  MoveL (T19476) to (113.08, 116.67, 20.1) mm, rotated rx 180 ry 0 rz -180 deg; joints [1.844, 67.674, -31.296, 3.106, -36.419, -2.5]
  Call Extruder 0.32811
  MoveL (T19477) to (108.19, 107.08, 20.1) mm, rotated rx 180 ry 0 rz -180 deg; joints [1.415, 68.728, -33.274, 2.439, -35.479, -1.986]
  Call Extruder 0.03668
  MoveL (T19478) to (108.19, 105.88, 20.1) mm, rotated rx 180 ry 0 rz -180 deg; joints [1.415, 68.728, -33.274, 2.439, -35.479, -1.986]
  Call Extruder 0.02276
  MoveL (T19479) to (108.94, 105.88, 20.1) mm, rotated rx 180 ry 0 rz -180 deg; joints [1.417, 68.56, -32.958, 2.433, -35.626, -1.978]
  Set speed (150.0 mm/s)
  MoveL (T19480) to (108.6, 106.28, 20.1) mm, rotated rx 180 ry 0 rz -180 deg; joints [1.417, 68.56, -32.958, 2.433, -35.626, -1.978]
  Set speed (25.0 mm/s)
  MoveL (T19481) to (108.6, 106.28, 20.1) mm, rotated rx 180 ry 0 rz -180 deg; joints [1.846, 67.513, -30.993, 3.099, -36.56, -2.49]
  Call Extruder 0.25102
  MoveL (T19482) to (116.84, 106.28, 20.1) mm, rotated rx 180 ry 0 rz -180 deg; joints [1.846, 67.513, -30.993, 3.099, -36.56, -2.49]
  Call Extruder 0.05979
  MoveL (T19483) to (116.84, 108.25, 20.1) mm, rotated rx 180 ry 0 rz -180 deg; joints [1.848, 67.353, -30.693, 3.093, -36.7, -2.48]
  Call Extruder 0.16307
  MoveL (T19484) to (111.48, 108.25, 20.1) mm, rotated rx 180 ry 0 rz -180 deg; joints [1.848, 67.353, -30.693, 3.093, -36.7, -2.48]
  Call Extruder 0.3456
  MoveL (T19485) to (116.65, 118.34, 20.1) mm, rotated rx 180 ry 0 rz -180 deg; joints [1.848, 67.353, -30.693, 3.093, -36.7, -2.48]
  Call Extruder 0.02131
  MoveL (T19486) to (116.65, 119.04, 20.1) mm, rotated rx 180 ry 0 rz -180 deg; joints [1.418, 68.393, -32.645, 2.427, -35.772, -1.969]
  Call Extruder 0.24283
  MoveL (T19487) to (108.68, 119.04, 20.1) mm, rotated rx 180 ry 0 rz -180 deg; joints [1.418, 68.393, -32.645, 2.427, -35.772, -1.969]
  Call Extruder 0.05979
  MoveL (T19488) to (108.68, 117.08, 20.1) mm, rotated rx 180 ry 0 rz -180 deg; joints [1.418, 68.393, -32.645, 2.427, -35.772, -1.969]
  Call Extruder 0.15438
  MoveL (T19489) to (113.75, 117.08, 20.1) mm, rotated rx 180 ry 0 rz -180 deg; joints [1.42, 68.227, -32.334, 2.421, -35.918, -1.961]
  Call Extruder 0.34538
  MoveL (T19490) to (108.6, 106.98, 20.1) mm, rotated rx 180 ry 0 rz -180 deg; joints [1.42, 68.227, -32.334, 2.421, -35.918, -1.961]
  Call Extruder 0.01947
  MoveL (T19491) to (108.6, 106.34, 20.1) mm, rotated rx 180 ry 0 rz -180 deg; joints [1.42, 68.227, -32.334, 2.421, -35.918, -1.961]
  Set speed (150.0 mm/s)
  MoveL (T19492) to (108.54, 105.89, 20.1) mm, rotated rx 180 ry 0 rz -180 deg; joints [1.85, 67.194, -30.394, 3.086, -36.84, -2.471]
  Set speed (45.0 mm/s)
  Call Extruder -1.6
  MoveL (T19493) to (108.54, 105.89, 20.1) mm, rotated rx 180 ry 0 rz -180 deg; joints [1.85, 67.194, -30.394, 3.086, -36.84, -2.471]
  Set speed (120.0 mm/s)
  MoveL (T19494) to (108.54, 105.89, 20.1) mm, rotated rx 180 ry 0 rz -180 deg; joints [1.85, 67.194, -30.394, 3.086, -36.84, -2.471]
  Call Extruder -0.38
  MoveL (T19495) to (109.66, 106.33, 20.1) mm, rotated rx 180 ry 0 rz -180 deg; joints [1.852, 67.036, -30.097, 3.08, -36.979, -2.461]
  Set speed (45.0 mm/s)
  Call Extruder -0.02
  MoveL (T19496) to (109.66, 106.33, 20.1) mm, rotated rx 180 ry 0 rz -180 deg; joints [1.852, 67.036, -30.097, 3.08, -36.979, -2.461]
  Set speed (150.0 mm/s)
  MoveL (T19497) to (109.66, 106.33, 22.1) mm, rotated rx 180 ry 0 rz -180 deg; joints [1.852, 67.036, -30.097, 3.08, -36.979, -2.461]
  MoveL (T19498) to (104.34, 103.54, 22.1) mm, rotated rx 180 ry 0 rz -180 deg; joints [1.422, 68.063, -32.025, 2.415, -36.062, -1.953]
  MoveL (T19499) to (104.34, 103.54, 20.1) mm, rotated rx 180 ry 0 rz -180 deg; joints [1.422, 68.063, -32.025, 2.415, -36.062, -1.953]
  Set speed (40.0 mm/s)
  Call Extruder 2.0
  MoveL (T19500) to (104.34, 103.54, 20.1) mm, rotated rx 180 ry 0 rz -180 deg; joints [1.422, 68.063, -32.025, 2.415, -36.062, -1.953]
  Call Extruder 0.52159
  MoveL (T19501) to (121.46, 103.54, 20.1) mm, rotated rx 180 ry 0 rz -180 deg; joints [1.423, 67.899, -31.717, 2.41, -36.206, -1.945]
  Call Extruder 0.54596
  MoveL (T19502) to (121.46, 121.46, 20.1) mm, rotated rx 180 ry 0 rz -180 deg; joints [1.854, 66.879, -29.802, 3.073, -37.117, -2.451]
  Call Extruder 0.54596
  MoveL (T19503) to (103.54, 121.46, 20.1) mm, rotated rx 180 ry 0 rz -180 deg; joints [1.854, 66.879, -29.802, 3.073, -37.117, -2.451]
  Call Extruder 0.54596
  MoveL (T19504) to (103.54, 103.54, 20.1) mm, rotated rx 180 ry 0 rz -180 deg; joints [1.856, 66.722, -29.509, 3.067, -37.253, -2.442]
  Call Extruder 0.02254
  MoveL (T19505) to (104.28, 103.54, 20.1) mm, rotated rx 180 ry 0 rz -180 deg; joints [1.856, 66.722, -29.509, 3.067, -37.253, -2.442]
  Set speed (150.0 mm/s)
  MoveL (T19506) to (103.53, 103.13, 20.1) mm, rotated rx 180 ry 0 rz -180 deg; joints [1.856, 66.722, -29.509, 3.067, -37.253, -2.442]
  Set speed (40.0 mm/s)
  MoveL (T19507) to (103.53, 103.13, 20.1) mm, rotated rx 180 ry 0 rz -180 deg; joints [1.425, 67.737, -31.412, 2.404, -36.348, -1.937]
  Call Extruder 0.55858
  MoveL (T19508) to (121.87, 103.13, 20.1) mm, rotated rx 180 ry 0 rz -180 deg; joints [1.425, 67.737, -31.412, 2.404, -36.348, -1.937]
  Call Extruder 0.57077
  MoveL (T19509) to (121.87, 121.87, 20.1) mm, rotated rx 180 ry 0 rz -180 deg; joints [1.425, 67.737, -31.412, 2.404, -36.348, -1.937]
  Call Extruder 0.57077
  MoveL (T19510) to (103.13, 121.87, 20.1) mm, rotated rx 180 ry 0 rz -180 deg; joints [1.425, 67.737, -31.412, 2.404, -36.348, -1.937]
  Call Extruder 0.57077
  MoveL (T19511) to (103.13, 103.13, 20.1) mm, rotated rx 180 ry 0 rz -180 deg; joints [1.426, 67.575, -31.109, 2.399, -36.49, -1.929]
  Call Extruder 0.01036
  MoveL (T19512) to (103.47, 103.13, 20.1) mm, rotated rx 180 ry 0 rz -180 deg; joints [1.426, 67.575, -31.109, 2.399, -36.49, -1.929]
  Set speed (150.0 mm/s)
  MoveL (T19513) to (102.72, 102.81, 20.1) mm, rotated rx 180 ry 0 rz -180 deg; joints [1.827, 66.638, -29.35, 3.014, -37.326, -2.397]
  Set speed (25.0 mm/s)
  MoveL (T19514) to (102.72, 102.81, 20.1) mm, rotated rx 180 ry 0 rz -180 deg; joints [1.827, 66.638, -29.35, 3.014, -37.326, -2.397]
  Call Extruder 0.00259
  MoveL (T19515) to (102.72, 102.72, 20.1) mm, rotated rx 180 ry 0 rz -180 deg; joints [1.827, 66.638, -29.35, 3.014, -37.326, -2.397]
  Call Extruder 0.59557
  MoveL (T19516) to (122.28, 102.72, 20.1) mm, rotated rx 180 ry 0 rz -180 deg; joints [1.796, 66.558, -29.2, 2.958, -37.395, -2.351]
  Call Extruder 0.59557
  MoveL (T19517) to (122.28, 122.28, 20.1) mm, rotated rx 180 ry 0 rz -180 deg; joints [1.796, 66.558, -29.2, 2.958, -37.395, -2.351]
  Call Extruder 0.59557
  MoveL (T19518) to (102.72, 122.28, 20.1) mm, rotated rx 180 ry 0 rz -180 deg; joints [1.796, 66.558, -29.2, 2.958, -37.395, -2.351]
  Call Extruder 0.59115
  MoveL (T19519) to (102.72, 102.87, 20.1) mm, rotated rx 180 ry 0 rz -180 deg; joints [1.428, 67.414, -30.808, 2.394, -36.631, -1.921]
  Set speed (150.0 mm/s)
  MoveL (T19520) to (102.78, 102.75, 20.1) mm, rotated rx 180 ry 0 rz -180 deg; joints [1.428, 67.414, -30.808, 2.394, -36.631, -1.921]
  Set speed (45.0 mm/s)
  Call Extruder -1.6
  MoveL (T19521) to (102.78, 102.75, 20.1) mm, rotated rx 180 ry 0 rz -180 deg; joints [1.429, 67.255, -30.508, 2.388, -36.771, -1.914]
  Set speed (120.0 mm/s)
  MoveL (T19522) to (102.78, 102.75, 20.1) mm, rotated rx 180 ry 0 rz -180 deg; joints [1.429, 67.255, -30.508, 2.388, -36.771, -1.914]
  Call Extruder -0.05166
  MoveL (T19523) to (102.72, 102.72, 20.1) mm, rotated rx 180 ry 0 rz -180 deg; joints [1.429, 67.255, -30.508, 2.388, -36.771, -1.914]
  Call Extruder -0.32834
  MoveL (T19524) to (103.65, 102.72, 20.1) mm, rotated rx 180 ry 0 rz -180 deg; joints [1.765, 66.478, -29.05, 2.902, -37.464, -2.304]
  Set speed (45.0 mm/s)
  Call Extruder -0.02
  MoveL (T19525) to (103.65, 102.72, 20.1) mm, rotated rx 180 ry 0 rz -180 deg; joints [1.765, 66.478, -29.05, 2.902, -37.464, -2.304]
  Set speed (150.0 mm/s)
  MoveL (T19526) to (103.65, 102.72, 22.1) mm, rotated rx 180 ry 0 rz -180 deg; joints [1.734, 66.398, -28.9, 2.846, -37.532, -2.258]
  MoveL (T19527) to (121.34, 120.62, 22.1) mm, rotated rx 180 ry 0 rz -180 deg; joints [1.431, 67.096, -30.21, 2.383, -36.91, -1.906]
  MoveL (T19528) to (121.34, 120.62, 20.1) mm, rotated rx 180 ry 0 rz -180 deg; joints [1.431, 67.096, -30.21, 2.383, -36.91, -1.906]
  Set speed (40.0 mm/s)
  Call Extruder 2.0
  MoveL (T19529) to (121.34, 120.62, 20.1) mm, rotated rx 180 ry 0 rz -180 deg; joints [1.431, 67.096, -30.21, 2.383, -36.91, -1.906]
  Set speed (25.0 mm/s)
  MoveL (T19530) to (121.34, 120.62, 20.1) mm, rotated rx 180 ry 0 rz -180 deg; joints [1.431, 67.096, -30.21, 2.383, -36.91, -1.906]
  Call Extruder 0.02133
  MoveL (T19531) to (120.78, 121.18, 20.1) mm, rotated rx 180 ry 0 rz -180 deg; joints [1.433, 66.939, -29.915, 2.378, -37.048, -1.899]
  Call Extruder 0.01356
  MoveL (T19532) to (120.27, 121.18, 20.1) mm, rotated rx 180 ry 0 rz -180 deg; joints [1.433, 66.939, -29.915, 2.378, -37.048, -1.899]
  Call Extruder 0.03442
  MoveL (T19533) to (121.18, 120.27, 20.1) mm, rotated rx 180 ry 0 rz -180 deg; joints [1.702, 66.319, -28.752, 2.791, -37.6, -2.212]
  Call Extruder 0.01356
  MoveL (T19534) to (121.18, 119.77, 20.1) mm, rotated rx 180 ry 0 rz -180 deg; joints [1.702, 66.319, -28.752, 2.791, -37.6, -2.212]
  Call Extruder 0.0536
  MoveL (T19535) to (119.77, 121.18, 20.1) mm, rotated rx 180 ry 0 rz -180 deg; joints [1.671, 66.24, -28.604, 2.736, -37.668, -2.166]
  Call Extruder 0.01356
  MoveL (T19536) to (119.26, 121.18, 20.1) mm, rotated rx 180 ry 0 rz -180 deg; joints [1.671, 66.24, -28.604, 2.736, -37.668, -2.166]
  Call Extruder 0.07278
  MoveL (T19537) to (121.18, 119.26, 20.1) mm, rotated rx 180 ry 0 rz -180 deg; joints [1.671, 66.24, -28.604, 2.736, -37.668, -2.166]
  Call Extruder 0.01356
  MoveL (T19538) to (121.18, 118.75, 20.1) mm, rotated rx 180 ry 0 rz -180 deg; joints [1.434, 66.782, -29.62, 2.373, -37.185, -1.891]
  Call Extruder 0.09196
  MoveL (T19539) to (118.75, 121.18, 20.1) mm, rotated rx 180 ry 0 rz -180 deg; joints [1.434, 66.782, -29.62, 2.373, -37.185, -1.891]
  Call Extruder 0.01356
  MoveL (T19540) to (118.25, 121.18, 20.1) mm, rotated rx 180 ry 0 rz -180 deg; joints [1.434, 66.782, -29.62, 2.373, -37.185, -1.891]
  Call Extruder 0.11113
  MoveL (T19541) to (121.18, 118.25, 20.1) mm, rotated rx 180 ry 0 rz -180 deg; joints [1.436, 66.626, -29.328, 2.369, -37.322, -1.884]
  Call Extruder 0.01356
  MoveL (T19542) to (121.18, 117.74, 20.1) mm, rotated rx 180 ry 0 rz -180 deg; joints [1.436, 66.626, -29.328, 2.369, -37.322, -1.884]
  Call Extruder 0.13031
  MoveL (T19543) to (117.74, 121.18, 20.1) mm, rotated rx 180 ry 0 rz -180 deg; joints [1.629, 66.186, -28.502, 2.664, -37.714, -2.108]
  Call Extruder 0.01356
  MoveL (T19544) to (117.23, 121.18, 20.1) mm, rotated rx 180 ry 0 rz -180 deg; joints [1.629, 66.186, -28.502, 2.664, -37.714, -2.108]
  Call Extruder 0.14949
  MoveL (T19545) to (121.18, 117.23, 20.1) mm, rotated rx 180 ry 0 rz -180 deg; joints [1.629, 66.186, -28.502, 2.664, -37.714, -2.108]
  Call Extruder 0.01356
  MoveL (T19546) to (121.18, 116.73, 20.1) mm, rotated rx 180 ry 0 rz -180 deg; joints [1.565, 66.182, -28.494, 2.559, -37.716, -2.025]
  Call Extruder 0.16867
  MoveL (T19547) to (116.73, 121.18, 20.1) mm, rotated rx 180 ry 0 rz -180 deg; joints [1.565, 66.182, -28.494, 2.559, -37.716, -2.025]
  Call Extruder 0.01356
  MoveL (T19548) to (116.22, 121.18, 20.1) mm, rotated rx 180 ry 0 rz -180 deg; joints [1.565, 66.182, -28.494, 2.559, -37.716, -2.025]
  Call Extruder 0.03951
  MoveL (T19549) to (117.27, 120.14, 20.1) mm, rotated rx 180 ry 0 rz -180 deg; joints [1.565, 66.182, -28.494, 2.559, -37.716, -2.025]
  Call Extruder 0.0129
  MoveL (T19550) to (117.75, 120.14, 20.1) mm, rotated rx 180 ry 0 rz -180 deg; joints [1.437, 66.471, -29.037, 2.364, -37.458, -1.877]
  Call Extruder 0.0129
  MoveL (T19551) to (117.75, 119.66, 20.1) mm, rotated rx 180 ry 0 rz -180 deg; joints [1.437, 66.471, -29.037, 2.364, -37.458, -1.877]
  Call Extruder 0.13009
  MoveL (T19552) to (121.18, 116.22, 20.1) mm, rotated rx 180 ry 0 rz -180 deg; joints [1.439, 66.317, -28.748, 2.359, -37.593, -1.87]
  Call Extruder 0.01356
  MoveL (T19553) to (121.18, 115.72, 20.1) mm, rotated rx 180 ry 0 rz -180 deg; joints [1.439, 66.317, -28.748, 2.359, -37.593, -1.87]
  Call Extruder 0.13009
  MoveL (T19554) to (117.75, 119.15, 20.1) mm, rotated rx 180 ry 0 rz -180 deg; joints [1.439, 66.317, -28.748, 2.359, -37.593, -1.87]
  Call Extruder 0.01356
  MoveL (T19555) to (117.75, 118.64, 20.1) mm, rotated rx 180 ry 0 rz -180 deg; joints [1.521, 66.132, -28.4, 2.485, -37.758, -1.965]
  Call Extruder 0.13009
  MoveL (T19556) to (121.18, 115.21, 20.1) mm, rotated rx 180 ry 0 rz -180 deg; joints [1.521, 66.132, -28.4, 2.485, -37.758, -1.965]
  Call Extruder 0.01356
  MoveL (T19557) to (121.18, 114.7, 20.1) mm, rotated rx 180 ry 0 rz -180 deg; joints [1.521, 66.132, -28.4, 2.485, -37.758, -1.965]
  Call Extruder 0.13009
  MoveL (T19558) to (117.75, 118.14, 20.1) mm, rotated rx 180 ry 0 rz -180 deg; joints [1.521, 66.132, -28.4, 2.485, -37.758, -1.965]
  Call Extruder 0.00153
  MoveL (T19559) to (117.75, 118.08, 20.1) mm, rotated rx 180 ry 0 rz -180 deg; joints [1.521, 66.132, -28.4, 2.485, -37.758, -1.965]
  Call Extruder 0.00894
  MoveL (T19560) to (117.59, 117.78, 20.1) mm, rotated rx 180 ry 0 rz -180 deg; joints [1.521, 66.132, -28.4, 2.485, -37.758, -1.965]
  Call Extruder 0.13584
  MoveL (T19561) to (121.18, 114.2, 20.1) mm, rotated rx 180 ry 0 rz -180 deg; joints [1.521, 66.132, -28.4, 2.485, -37.758, -1.965]
  Call Extruder 0.01356
  MoveL (T19562) to (121.18, 113.69, 20.1) mm, rotated rx 180 ry 0 rz -180 deg; joints [1.521, 66.132, -28.4, 2.485, -37.758, -1.965]
  Call Extruder 0.14234
  MoveL (T19563) to (117.42, 117.45, 20.1) mm, rotated rx 180 ry 0 rz -180 deg; joints [1.521, 66.132, -28.4, 2.485, -37.758, -1.965]
  Call Extruder 0.01008
  MoveL (T19564) to (117.25, 117.11, 20.1) mm, rotated rx 180 ry 0 rz -180 deg; joints [1.521, 66.132, -28.4, 2.485, -37.758, -1.965]
  Call Extruder 0.14883
  MoveL (T19565) to (121.18, 113.19, 20.1) mm, rotated rx 180 ry 0 rz -180 deg; joints [1.521, 66.132, -28.4, 2.485, -37.758, -1.965]
  Call Extruder 0.01356
  MoveL (T19566) to (121.18, 112.68, 20.1) mm, rotated rx 180 ry 0 rz -180 deg; joints [1.521, 66.132, -28.4, 2.485, -37.758, -1.965]
  Call Extruder 0.15532
  MoveL (T19567) to (117.08, 116.78, 20.1) mm, rotated rx 180 ry 0 rz -180 deg; joints [1.439, 66.317, -28.748, 2.359, -37.593, -1.87]
  Call Extruder 0.01008
  MoveL (T19568) to (116.91, 116.44, 20.1) mm, rotated rx 180 ry 0 rz -180 deg; joints [1.439, 66.317, -28.748, 2.359, -37.593, -1.87]
  Call Extruder 0.16181
  MoveL (T19569) to (121.18, 112.17, 20.1) mm, rotated rx 180 ry 0 rz -180 deg; joints [1.439, 66.317, -28.748, 2.359, -37.593, -1.87]
  Call Extruder 0.01356
  MoveL (T19570) to (121.18, 111.67, 20.1) mm, rotated rx 180 ry 0 rz -180 deg; joints [1.439, 66.323, -28.759, 2.36, -37.588, -1.87]
  Call Extruder 0.1683
  MoveL (T19571) to (116.74, 116.11, 20.1) mm, rotated rx 180 ry 0 rz -180 deg; joints [1.439, 66.323, -28.759, 2.36, -37.588, -1.87]
  Call Extruder 0.01008
  MoveL (T19572) to (116.57, 115.77, 20.1) mm, rotated rx 180 ry 0 rz -180 deg; joints [1.439, 66.323, -28.759, 2.36, -37.588, -1.87]
  Call Extruder 0.1748
  MoveL (T19573) to (121.18, 111.16, 20.1) mm, rotated rx 180 ry 0 rz -180 deg; joints [1.439, 66.323, -28.759, 2.36, -37.588, -1.87]
  Call Extruder 0.01356
  MoveL (T19574) to (121.18, 110.65, 20.1) mm, rotated rx 180 ry 0 rz -180 deg; joints [1.439, 66.323, -28.759, 2.36, -37.588, -1.87]
  Call Extruder 0.18129
  MoveL (T19575) to (116.39, 115.44, 20.1) mm, rotated rx 180 ry 0 rz -180 deg; joints [1.439, 66.323, -28.759, 2.36, -37.588, -1.87]
  Call Extruder 0.01008
  MoveL (T19576) to (116.22, 115.1, 20.1) mm, rotated rx 180 ry 0 rz -180 deg; joints [1.439, 66.323, -28.759, 2.36, -37.588, -1.87]
  Call Extruder 0.18778
  MoveL (T19577) to (121.18, 110.15, 20.1) mm, rotated rx 180 ry 0 rz -180 deg; joints [1.888, 67.418, -31.218, 3.194, -36.243, -2.577]
  Call Extruder 0.01356
  MoveL (T19578) to (121.18, 109.64, 20.1) mm, rotated rx 180 ry 0 rz -180 deg; joints [1.888, 67.418, -31.218, 3.194, -36.243, -2.577]
  Call Extruder 0.19427
  MoveL (T19579) to (116.05, 114.77, 20.1) mm, rotated rx 180 ry 0 rz -180 deg; joints [1.888, 67.652, -31.254, 3.179, -36.44, -2.558]
  Call Extruder 0.01008
  MoveL (T19580) to (115.88, 114.43, 20.1) mm, rotated rx 180 ry 0 rz -180 deg; joints [1.888, 67.652, -31.254, 3.179, -36.44, -2.558]
  Call Extruder 0.20076
  MoveL (T19581) to (121.18, 109.14, 20.1) mm, rotated rx 180 ry 0 rz -180 deg; joints [1.888, 67.652, -31.254, 3.179, -36.44, -2.558]
  Call Extruder 0.01356
  MoveL (T19582) to (121.18, 108.63, 20.1) mm, rotated rx 180 ry 0 rz -180 deg; joints [1.888, 67.652, -31.254, 3.179, -36.44, -2.558]
  Call Extruder 0.20726
  MoveL (T19583) to (115.71, 114.1, 20.1) mm, rotated rx 180 ry 0 rz -180 deg; joints [1.888, 67.652, -31.254, 3.179, -36.44, -2.558]
  Call Extruder 0.01008
  MoveL (T19584) to (115.54, 113.77, 20.1) mm, rotated rx 180 ry 0 rz -180 deg; joints [1.888, 67.652, -31.254, 3.179, -36.44, -2.558]
  Call Extruder 0.21375
  MoveL (T19585) to (121.18, 108.12, 20.1) mm, rotated rx 180 ry 0 rz -180 deg; joints [1.888, 67.652, -31.254, 3.179, -36.44, -2.558]
  Call Extruder 0.01356
  MoveL (T19586) to (121.18, 107.62, 20.1) mm, rotated rx 180 ry 0 rz -180 deg; joints [1.888, 67.652, -31.254, 3.179, -36.44, -2.558]
  Call Extruder 0.22024
  MoveL (T19587) to (115.37, 113.43, 20.1) mm, rotated rx 180 ry 0 rz -180 deg; joints [1.888, 67.652, -31.254, 3.179, -36.44, -2.558]
  Call Extruder 0.01008
  MoveL (T19588) to (115.2, 113.09, 20.1) mm, rotated rx 180 ry 0 rz -180 deg; joints [1.888, 67.652, -31.254, 3.179, -36.44, -2.558]
  Call Extruder 0.22673
  MoveL (T19589) to (121.18, 107.11, 20.1) mm, rotated rx 180 ry 0 rz -180 deg; joints [1.884, 67.911, -31.74, 3.19, -36.213, -2.575]
  Call Extruder 0.01356
  MoveL (T19590) to (121.18, 106.6, 20.1) mm, rotated rx 180 ry 0 rz -180 deg; joints [1.884, 67.911, -31.74, 3.19, -36.213, -2.575]
  Call Extruder 0.23322
  MoveL (T19591) to (115.02, 112.76, 20.1) mm, rotated rx 180 ry 0 rz -180 deg; joints [1.875, 67.966, -31.843, 3.178, -36.165, -2.566]
  Call Extruder 0.01008
  MoveL (T19592) to (114.85, 112.42, 20.1) mm, rotated rx 180 ry 0 rz -180 deg; joints [1.875, 67.966, -31.843, 3.178, -36.165, -2.566]
  Call Extruder 0.23972
  MoveL (T19593) to (121.18, 106.1, 20.1) mm, rotated rx 180 ry 0 rz -180 deg; joints [1.875, 67.966, -31.843, 3.178, -36.165, -2.566]
  Call Extruder 0.01356
  MoveL (T19594) to (121.18, 105.59, 20.1) mm, rotated rx 180 ry 0 rz -180 deg; joints [1.775, 68.208, -32.297, 3.024, -35.949, -2.449]
  Call Extruder 0.12308
  MoveL (T19595) to (117.93, 108.84, 20.1) mm, rotated rx 180 ry 0 rz -180 deg; joints [1.775, 68.208, -32.297, 3.024, -35.949, -2.449]
  Call Extruder 0.01337
  MoveL (T19596) to (117.93, 109.34, 20.1) mm, rotated rx 180 ry 0 rz -180 deg; joints [2.29, 69.699, -35.098, 4.028, -34.668, -3.315]
  Call Extruder 0.01337
  MoveL (T19597) to (117.43, 109.34, 20.1) mm, rotated rx 180 ry 0 rz -180 deg; joints [2.29, 69.699, -35.098, 4.028, -34.668, -3.315]
  Call Extruder 0.10422
  MoveL (T19598) to (114.68, 112.09, 20.1) mm, rotated rx 180 ry 0 rz -180 deg; joints [2.356, 69.707, -35.112, 4.144, -34.665, -3.41]
  Call Extruder 0.01008
  MoveL (T19599) to (114.51, 111.75, 20.1) mm, rotated rx 180 ry 0 rz -180 deg; joints [2.356, 69.707, -35.112, 4.144, -34.665, -3.41]
  Call Extruder 0.09153
  MoveL (T19600) to (116.93, 109.34, 20.1) mm, rotated rx 180 ry 0 rz -180 deg; joints [2.356, 69.707, -35.112, 4.144, -34.665, -3.41]
  Call Extruder 0.01356
  MoveL (T19601) to (116.42, 109.34, 20.1) mm, rotated rx 180 ry 0 rz -180 deg; joints [3.288, 67.468, -30.908, 5.508, -36.687, -4.422]
  Call Extruder 0.07885
  MoveL (T19602) to (114.34, 111.42, 20.1) mm, rotated rx 180 ry 0 rz -180 deg; joints [3.288, 67.468, -30.908, 5.508, -36.687, -4.422]
  Call Extruder 0.01008
  MoveL (T19603) to (114.17, 111.09, 20.1) mm, rotated rx 180 ry 0 rz -180 deg; joints [3.288, 67.468, -30.908, 5.508, -36.687, -4.422]
  Call Extruder 0.06616
  MoveL (T19604) to (115.91, 109.34, 20.1) mm, rotated rx 180 ry 0 rz -180 deg; joints [3.295, 67.17, -30.349, 5.486, -36.948, -4.389]
  Call Extruder 0.01356
  MoveL (T19605) to (115.41, 109.34, 20.1) mm, rotated rx 180 ry 0 rz -180 deg; joints [3.295, 67.17, -30.349, 5.486, -36.948, -4.389]
  Call Extruder 0.05348
  MoveL (T19606) to (114, 110.75, 20.1) mm, rotated rx 180 ry 0 rz -180 deg; joints [2.938, 66.204, -28.536, 4.801, -37.766, -3.799]
  Call Extruder 0.01008
  MoveL (T19607) to (113.83, 110.42, 20.1) mm, rotated rx 180 ry 0 rz -180 deg; joints [2.938, 66.204, -28.536, 4.801, -37.766, -3.799]
  Call Extruder 0.04079
  MoveL (T19608) to (114.9, 109.34, 20.1) mm, rotated rx 180 ry 0 rz -180 deg; joints [2.938, 66.204, -28.536, 4.801, -37.766, -3.799]
  Call Extruder 0.01356
  MoveL (T19609) to (114.39, 109.34, 20.1) mm, rotated rx 180 ry 0 rz -180 deg; joints [2.938, 66.204, -28.536, 4.801, -37.766, -3.799]
  Call Extruder 0.0281
  MoveL (T19610) to (113.65, 110.08, 20.1) mm, rotated rx 180 ry 0 rz -180 deg; joints [2.818, 66.19, -28.509, 4.604, -37.771, -3.642]
  Call Extruder 0.01008
  MoveL (T19611) to (113.48, 109.75, 20.1) mm, rotated rx 180 ry 0 rz -180 deg; joints [1.815, 68.507, -32.858, 3.112, -35.689, -2.528]
  Call Extruder 0.01542
  MoveL (T19612) to (113.89, 109.34, 20.1) mm, rotated rx 180 ry 0 rz -180 deg; joints [1.815, 68.507, -32.858, 3.112, -35.689, -2.528]
  Call Extruder 0.01356
  MoveL (T19613) to (113.38, 109.34, 20.1) mm, rotated rx 180 ry 0 rz -180 deg; joints [1.866, 68.651, -33.13, 3.21, -35.564, -2.612]
  Call Extruder 0.00725
  MoveL (T19614) to (113.19, 109.53, 20.1) mm, rotated rx 180 ry 0 rz -180 deg; joints [1.866, 68.651, -33.13, 3.21, -35.564, -2.612]
  Set speed (45.0 mm/s)
  Call Extruder -1.6
  MoveL (T19615) to (113.19, 109.53, 20.1) mm, rotated rx 180 ry 0 rz -180 deg; joints [1.866, 68.651, -33.13, 3.21, -35.564, -2.612]
  Set speed (120.0 mm/s)
  MoveL (T19616) to (113.19, 109.53, 20.1) mm, rotated rx 180 ry 0 rz -180 deg; joints [1.866, 68.651, -33.13, 3.21, -35.564, -2.612]
  Call Extruder -0.09648
  MoveL (T19617) to (113.38, 109.34, 20.1) mm, rotated rx 180 ry 0 rz -180 deg; joints [1.866, 68.651, -33.13, 3.21, -35.564, -2.612]
  Call Extruder -0.18035
  MoveL (T19618) to (113.89, 109.34, 20.1) mm, rotated rx 180 ry 0 rz -180 deg; joints [1.874, 68.709, -33.238, 3.228, -35.514, -2.628]
  Call Extruder -0.10317
  MoveL (T19619) to (113.68, 109.54, 20.1) mm, rotated rx 180 ry 0 rz -180 deg; joints [1.869, 69.145, -34.057, 3.249, -35.132, -2.658]
  Set speed (45.0 mm/s)
  Call Extruder -0.02
  MoveL (T19620) to (113.68, 109.54, 20.1) mm, rotated rx 180 ry 0 rz -180 deg; joints [1.869, 69.145, -34.057, 3.249, -35.132, -2.658]
  Set speed (150.0 mm/s)
  MoveL (T19621) to (113.68, 109.54, 22.1) mm, rotated rx 180 ry 0 rz -180 deg; joints [1.869, 69.145, -34.057, 3.249, -35.132, -2.658]
  MoveL (T19622) to (117.77, 108.5, 22.1) mm, rotated rx 180 ry 0 rz -180 deg; joints [1.869, 69.145, -34.057, 3.249, -35.132, -2.658]
  MoveL (T19623) to (117.77, 108.5, 20.1) mm, rotated rx 180 ry 0 rz -180 deg; joints [1.869, 69.145, -34.057, 3.249, -35.132, -2.658]
  Set speed (40.0 mm/s)
  Call Extruder 2.0
  MoveL (T19624) to (117.77, 108.5, 20.1) mm, rotated rx 180 ry 0 rz -180 deg; joints [1.869, 69.145, -34.057, 3.249, -35.132, -2.658]
  Set speed (25.0 mm/s)
  MoveL (T19625) to (117.77, 108.5, 20.1) mm, rotated rx 180 ry 0 rz -180 deg; joints [1.869, 69.145, -34.057, 3.249, -35.132, -2.658]
  Call Extruder 0.12917
  MoveL (T19626) to (121.18, 105.08, 20.1) mm, rotated rx 180 ry 0 rz -180 deg; joints [1.869, 69.145, -34.057, 3.249, -35.132, -2.658]
  Call Extruder 0.01356
  MoveL (T19627) to (121.18, 104.58, 20.1) mm, rotated rx 180 ry 0 rz -180 deg; joints [1.869, 69.145, -34.057, 3.249, -35.132, -2.658]
  Call Extruder 0.12308
  MoveL (T19628) to (117.93, 107.83, 20.1) mm, rotated rx 180 ry 0 rz -180 deg; joints [1.873, 68.839, -33.482, 3.234, -35.4, -2.637]
  Call Extruder 0.01356
  MoveL (T19629) to (117.93, 107.32, 20.1) mm, rotated rx 180 ry 0 rz -180 deg; joints [1.873, 68.839, -33.482, 3.234, -35.4, -2.637]
  Call Extruder 0.12308
  MoveL (T19630) to (121.18, 104.07, 20.1) mm, rotated rx 180 ry 0 rz -180 deg; joints [1.873, 68.839, -33.482, 3.234, -35.4, -2.637]
  Call Extruder 0.00678
  MoveL (T19631) to (121.18, 103.82, 20.1) mm, rotated rx 180 ry 0 rz -180 deg; joints [1.873, 68.839, -33.482, 3.234, -35.4, -2.637]
  Call Extruder 0.00678
  MoveL (T19632) to (120.93, 103.82, 20.1) mm, rotated rx 180 ry 0 rz -180 deg; joints [1.873, 68.839, -33.482, 3.234, -35.4, -2.637]
  Call Extruder 0.11349
  MoveL (T19633) to (117.93, 106.81, 20.1) mm, rotated rx 180 ry 0 rz -180 deg; joints [1.873, 68.839, -33.482, 3.234, -35.4, -2.637]
  Call Extruder 0.01356
  MoveL (T19634) to (117.93, 106.31, 20.1) mm, rotated rx 180 ry 0 rz -180 deg; joints [1.873, 68.605, -33.443, 3.249, -35.206, -2.656]
  Call Extruder 0.09431
  MoveL (T19635) to (120.42, 103.82, 20.1) mm, rotated rx 180 ry 0 rz -180 deg; joints [1.652, 70.731, -37.43, 3.008, -33.337, -2.513]
  Call Extruder 0.01356
  MoveL (T19636) to (119.92, 103.82, 20.1) mm, rotated rx 180 ry 0 rz -180 deg; joints [1.652, 70.963, -37.471, 2.993, -33.527, -2.495]
  Call Extruder 0.07513
  MoveL (T19637) to (117.93, 105.8, 20.1) mm, rotated rx 180 ry 0 rz -180 deg; joints [1.652, 70.963, -37.471, 2.993, -33.527, -2.495]
  Call Extruder 0.01356
  MoveL (T19638) to (117.93, 105.3, 20.1) mm, rotated rx 180 ry 0 rz -180 deg; joints [1.652, 70.963, -37.471, 2.993, -33.527, -2.495]
  Call Extruder 0.05596
  MoveL (T19639) to (119.41, 103.82, 20.1) mm, rotated rx 180 ry 0 rz -180 deg; joints [1.652, 70.963, -37.471, 2.993, -33.527, -2.495]
  Call Extruder 0.01356
  MoveL (T19640) to (118.9, 103.82, 20.1) mm, rotated rx 180 ry 0 rz -180 deg; joints [1.652, 70.963, -37.471, 2.993, -33.527, -2.495]
  Call Extruder 0.05183
  MoveL (T19641) to (117.53, 105.19, 20.1) mm, rotated rx 180 ry 0 rz -180 deg; joints [1.652, 70.963, -37.471, 2.993, -33.527, -2.495]
  Call Extruder 0.01356
  MoveL (T19642) to (117.03, 105.19, 20.1) mm, rotated rx 180 ry 0 rz -180 deg; joints [1.652, 70.963, -37.471, 2.993, -33.527, -2.495]
  Call Extruder 0.05183
  MoveL (T19643) to (118.4, 103.82, 20.1) mm, rotated rx 180 ry 0 rz -180 deg; joints [1.652, 70.963, -37.471, 2.993, -33.527, -2.495]
  Call Extruder 0.01356
  MoveL (T19644) to (117.89, 103.82, 20.1) mm, rotated rx 180 ry 0 rz -180 deg; joints [1.652, 70.963, -37.471, 2.993, -33.527, -2.495]
  Call Extruder 0.05183
  MoveL (T19645) to (116.52, 105.19, 20.1) mm, rotated rx 180 ry 0 rz -180 deg; joints [1.652, 70.963, -37.471, 2.993, -33.527, -2.495]
  Call Extruder 0.01356
  MoveL (T19646) to (116.02, 105.19, 20.1) mm, rotated rx 180 ry 0 rz -180 deg; joints [1.396, 70.942, -37.433, 2.527, -33.535, -2.107]
  Call Extruder 0.05183
  MoveL (T19647) to (117.38, 103.82, 20.1) mm, rotated rx 180 ry 0 rz -180 deg; joints [1.396, 70.942, -37.433, 2.527, -33.535, -2.107]
  Call Extruder 0.01356
  MoveL (T19648) to (116.88, 103.82, 20.1) mm, rotated rx 180 ry 0 rz -180 deg; joints [1.467, 70.743, -37.059, 2.643, -33.712, -2.199]
  Call Extruder 0.05183
  MoveL (T19649) to (115.51, 105.19, 20.1) mm, rotated rx 180 ry 0 rz -180 deg; joints [1.467, 70.743, -37.059, 2.643, -33.712, -2.199]
  Call Extruder 0.01356
  MoveL (T19650) to (115, 105.19, 20.1) mm, rotated rx 180 ry 0 rz -180 deg; joints [1.467, 70.743, -37.059, 2.643, -33.712, -2.199]
  Call Extruder 0.05183
  MoveL (T19651) to (116.37, 103.82, 20.1) mm, rotated rx 180 ry 0 rz -180 deg; joints [1.607, 70.754, -37.08, 2.896, -33.708, -2.41]
  Call Extruder 0.01356
  MoveL (T19652) to (115.86, 103.82, 20.1) mm, rotated rx 180 ry 0 rz -180 deg; joints [1.607, 70.754, -37.08, 2.896, -33.708, -2.41]
  Call Extruder 0.05183
  MoveL (T19653) to (114.5, 105.19, 20.1) mm, rotated rx 180 ry 0 rz -180 deg; joints [1.628, 70.73, -37.035, 2.933, -33.73, -2.44]
  Call Extruder 0.01356
  MoveL (T19654) to (113.99, 105.19, 20.1) mm, rotated rx 180 ry 0 rz -180 deg; joints [1.628, 70.73, -37.035, 2.933, -33.73, -2.44]
  Call Extruder 0.05183
  MoveL (T19655) to (115.36, 103.82, 20.1) mm, rotated rx 180 ry 0 rz -180 deg; joints [1.628, 70.73, -37.035, 2.933, -33.73, -2.44]
  Call Extruder 0.01356
  MoveL (T19656) to (114.85, 103.82, 20.1) mm, rotated rx 180 ry 0 rz -180 deg; joints [1.659, 70.645, -36.875, 2.982, -33.806, -2.478]
  Call Extruder 0.05183
  MoveL (T19657) to (113.48, 105.19, 20.1) mm, rotated rx 180 ry 0 rz -180 deg; joints [1.659, 70.645, -36.875, 2.982, -33.806, -2.478]
  Call Extruder 0.01356
  MoveL (T19658) to (112.98, 105.19, 20.1) mm, rotated rx 180 ry 0 rz -180 deg; joints [1.659, 70.645, -36.875, 2.982, -33.806, -2.478]
  Call Extruder 0.05183
  MoveL (T19659) to (114.35, 103.82, 20.1) mm, rotated rx 180 ry 0 rz -180 deg; joints [1.763, 70.972, -37.49, 3.193, -33.524, -2.663]
  Call Extruder 0.01356
  MoveL (T19660) to (113.84, 103.82, 20.1) mm, rotated rx 180 ry 0 rz -180 deg; joints [1.763, 70.972, -37.49, 3.193, -33.524, -2.663]
  Call Extruder 0.05183
  MoveL (T19661) to (112.47, 105.19, 20.1) mm, rotated rx 180 ry 0 rz -180 deg; joints [1.787, 70.975, -37.494, 3.237, -33.523, -2.699]
  Call Extruder 0.01356
  MoveL (T19662) to (111.97, 105.19, 20.1) mm, rotated rx 180 ry 0 rz -180 deg; joints [1.787, 70.975, -37.494, 3.237, -33.523, -2.699]
  Call Extruder 0.05183
  MoveL (T19663) to (113.33, 103.82, 20.1) mm, rotated rx 180 ry 0 rz -180 deg; joints [1.787, 70.975, -37.494, 3.237, -33.523, -2.699]
  Call Extruder 0.01356
  MoveL (T19664) to (112.83, 103.82, 20.1) mm, rotated rx 180 ry 0 rz -180 deg; joints [1.794, 70.346, -36.313, 3.202, -34.075, -2.653]
  Call Extruder 0.05183
  MoveL (T19665) to (111.46, 105.19, 20.1) mm, rotated rx 180 ry 0 rz -180 deg; joints [1.794, 70.346, -36.313, 3.202, -34.075, -2.653]
  Call Extruder 0.01356
  MoveL (T19666) to (110.95, 105.19, 20.1) mm, rotated rx 180 ry 0 rz -180 deg; joints [1.803, 70.286, -36.199, 3.215, -34.128, -2.662]
  Call Extruder 0.05183
  MoveL (T19667) to (112.32, 103.82, 20.1) mm, rotated rx 180 ry 0 rz -180 deg; joints [1.803, 70.286, -36.199, 3.215, -34.128, -2.662]
  Call Extruder 0.01356
  MoveL (T19668) to (111.81, 103.82, 20.1) mm, rotated rx 180 ry 0 rz -180 deg; joints [1.803, 70.286, -36.199, 3.215, -34.128, -2.662]
  Call Extruder 0.05183
  MoveL (T19669) to (110.45, 105.19, 20.1) mm, rotated rx 180 ry 0 rz -180 deg; joints [1.803, 70.286, -36.199, 3.215, -34.128, -2.662]
  Call Extruder 0.01356
  MoveL (T19670) to (109.94, 105.19, 20.1) mm, rotated rx 180 ry 0 rz -180 deg; joints [1.803, 70.286, -36.199, 3.215, -34.128, -2.662]
  Call Extruder 0.05183
  MoveL (T19671) to (111.31, 103.82, 20.1) mm, rotated rx 180 ry 0 rz -180 deg; joints [1.915, 69.986, -35.637, 3.391, -34.396, -2.799]
  Call Extruder 0.01356
  MoveL (T19672) to (110.8, 103.82, 20.1) mm, rotated rx 180 ry 0 rz -180 deg; joints [1.915, 69.986, -35.637, 3.391, -34.396, -2.799]
  Call Extruder 0.05183
  MoveL (T19673) to (109.44, 105.19, 20.1) mm, rotated rx 180 ry 0 rz -180 deg; joints [1.915, 69.986, -35.637, 3.391, -34.396, -2.799]
  Call Extruder 0.01356
  MoveL (T19674) to (108.93, 105.19, 20.1) mm, rotated rx 180 ry 0 rz -180 deg; joints [1.915, 69.986, -35.637, 3.391, -34.396, -2.799]
  Call Extruder 0.05183
  MoveL (T19675) to (110.3, 103.82, 20.1) mm, rotated rx 180 ry 0 rz -180 deg; joints [1.861, 69.824, -35.332, 3.284, -34.536, -2.706]
  Call Extruder 0.01356
  MoveL (T19676) to (109.79, 103.82, 20.1) mm, rotated rx 180 ry 0 rz -180 deg; joints [1.863, 69.672, -35.047, 3.276, -34.669, -2.695]
  Call Extruder 0.05792
  MoveL (T19677) to (108.26, 105.35, 20.1) mm, rotated rx 180 ry 0 rz -180 deg; joints [1.863, 69.672, -35.047, 3.276, -34.669, -2.695]
  Set speed (45.0 mm/s)
  Call Extruder -1.6
  MoveL (T19678) to (108.26, 105.35, 20.1) mm, rotated rx 180 ry 0 rz -180 deg; joints [3.316, 66.253, -28.628, 5.422, -37.75, -4.292]
  Set speed (120.0 mm/s)
  MoveL (T19679) to (108.26, 105.35, 20.1) mm, rotated rx 180 ry 0 rz -180 deg; joints [3.316, 66.253, -28.628, 5.422, -37.75, -4.292]
  Call Extruder -0.38
  MoveL (T19680) to (109.02, 104.59, 20.1) mm, rotated rx 180 ry 0 rz -180 deg; joints [3.301, 66.891, -29.824, 5.466, -37.192, -4.359]
  Set speed (45.0 mm/s)
  Call Extruder -0.02
  MoveL (T19681) to (109.02, 104.59, 20.1) mm, rotated rx 180 ry 0 rz -180 deg; joints [3.301, 66.891, -29.824, 5.466, -37.192, -4.359]
  Set speed (150.0 mm/s)
  MoveL (T19682) to (109.02, 104.59, 22.1) mm, rotated rx 180 ry 0 rz -180 deg; joints [3.301, 66.891, -29.824, 5.466, -37.192, -4.359]
  MoveL (T19683) to (112.03, 115.76, 22.1) mm, rotated rx 180 ry 0 rz -180 deg; joints [3.301, 66.891, -29.824, 5.466, -37.192, -4.359]
  MoveL (T19684) to (112.03, 115.76, 20.1) mm, rotated rx 180 ry 0 rz -180 deg; joints [3.301, 66.891, -29.824, 5.466, -37.192, -4.359]
  Set speed (40.0 mm/s)
  Call Extruder 2.0
  MoveL (T19685) to (112.03, 115.76, 20.1) mm, rotated rx 180 ry 0 rz -180 deg; joints [3.301, 66.891, -29.824, 5.466, -37.192, -4.359]
  Set speed (25.0 mm/s)
  MoveL (T19686) to (112.03, 115.76, 20.1) mm, rotated rx 180 ry 0 rz -180 deg; joints [3.301, 66.891, -29.824, 5.466, -37.192, -4.359]
  Call Extruder 0.00864
  MoveL (T19687) to (111.8, 115.99, 20.1) mm, rotated rx 180 ry 0 rz -180 deg; joints [3.301, 66.891, -29.824, 5.466, -37.192, -4.359]
  Call Extruder 0.01356
  MoveL (T19688) to (111.29, 115.99, 20.1) mm, rotated rx 180 ry 0 rz -180 deg; joints [3.301, 66.891, -29.824, 5.466, -37.192, -4.359]
  Call Extruder 0.01681
  MoveL (T19689) to (111.74, 115.54, 20.1) mm, rotated rx 180 ry 0 rz -180 deg; joints [3.308, 66.61, -29.298, 5.446, -37.437, -4.329]
  Call Extruder 0.01008
  MoveL (T19690) to (111.56, 115.21, 20.1) mm, rotated rx 180 ry 0 rz -180 deg; joints [3.308, 66.61, -29.298, 5.446, -37.437, -4.329]
  Call Extruder 0.02951
  MoveL (T19691) to (110.79, 115.99, 20.1) mm, rotated rx 180 ry 0 rz -180 deg; joints [3.308, 66.61, -29.298, 5.446, -37.437, -4.329]
  Call Extruder 0.01356
  MoveL (T19692) to (110.28, 115.99, 20.1) mm, rotated rx 180 ry 0 rz -180 deg; joints [3.308, 66.61, -29.298, 5.446, -37.437, -4.329]
  Call Extruder 0.04221
  MoveL (T19693) to (111.39, 114.87, 20.1) mm, rotated rx 180 ry 0 rz -180 deg; joints [3.308, 66.61, -29.298, 5.446, -37.437, -4.329]
  Call Extruder 0.01008
  MoveL (T19694) to (111.22, 114.54, 20.1) mm, rotated rx 180 ry 0 rz -180 deg; joints [3.308, 66.61, -29.298, 5.446, -37.437, -4.329]
  Call Extruder 0.05491
  MoveL (T19695) to (109.77, 115.99, 20.1) mm, rotated rx 180 ry 0 rz -180 deg; joints [1.407, 65.958, -28.481, 2.312, -37.5, -1.835]
  Call Extruder 0.01356
  MoveL (T19696) to (109.27, 115.99, 20.1) mm, rotated rx 180 ry 0 rz -180 deg; joints [1.407, 66.17, -28.512, 2.303, -37.68, -1.823]
  Call Extruder 0.06761
  MoveL (T19697) to (111.05, 114.2, 20.1) mm, rotated rx 180 ry 0 rz -180 deg; joints [1.407, 66.17, -28.512, 2.303, -37.68, -1.823]
  Call Extruder 0.01008
  MoveL (T19698) to (110.88, 113.87, 20.1) mm, rotated rx 180 ry 0 rz -180 deg; joints [1.407, 66.17, -28.512, 2.303, -37.68, -1.823]
  Call Extruder 0.08031
  MoveL (T19699) to (108.76, 115.99, 20.1) mm, rotated rx 180 ry 0 rz -180 deg; joints [1.407, 66.17, -28.512, 2.303, -37.68, -1.823]
  Call Extruder 0.01356
  MoveL (T19700) to (108.25, 115.99, 20.1) mm, rotated rx 180 ry 0 rz -180 deg; joints [1.407, 66.17, -28.512, 2.303, -37.68, -1.823]
  Call Extruder 0.09754
  MoveL (T19701) to (110.83, 113.41, 20.1) mm, rotated rx 180 ry 0 rz -180 deg; joints [1.407, 66.17, -28.512, 2.303, -37.68, -1.823]
  Set speed (45.0 mm/s)
  Call Extruder -1.6
  MoveL (T19702) to (110.83, 113.41, 20.1) mm, rotated rx 180 ry 0 rz -180 deg; joints [1.407, 66.17, -28.512, 2.303, -37.68, -1.823]
  Set speed (120.0 mm/s)
  MoveL (T19703) to (110.83, 113.41, 20.1) mm, rotated rx 180 ry 0 rz -180 deg; joints [1.363, 71.012, -37.604, 2.475, -33.433, -2.066]
  Call Extruder -0.38
  MoveL (T19704) to (110.08, 114.17, 20.1) mm, rotated rx 180 ry 0 rz -180 deg; joints [1.363, 71.012, -37.604, 2.475, -33.433, -2.066]
  Set speed (45.0 mm/s)
  Call Extruder -0.02
  MoveL (T19705) to (110.08, 114.17, 20.1) mm, rotated rx 180 ry 0 rz -180 deg; joints [3.241, 71.239, -38.03, 5.904, -33.349, -4.937]
  Set speed (150.0 mm/s)
  MoveL (T19706) to (110.08, 114.17, 22.1) mm, rotated rx 180 ry 0 rz -180 deg; joints [3.241, 71.239, -38.03, 5.904, -33.349, -4.937]
  MoveL (T19707) to (115.56, 121.34, 22.1) mm, rotated rx 180 ry 0 rz -180 deg; joints [3.241, 71.239, -38.03, 5.904, -33.349, -4.937]
  MoveL (T19708) to (115.56, 121.34, 20.1) mm, rotated rx 180 ry 0 rz -180 deg; joints [3.241, 71.239, -38.03, 5.904, -33.349, -4.937]
  Set speed (40.0 mm/s)
  Call Extruder 2.0
  MoveL (T19709) to (115.56, 121.34, 20.1) mm, rotated rx 180 ry 0 rz -180 deg; joints [3.351, 66.156, -28.485, 5.473, -37.797, -4.33]
  Set speed (25.0 mm/s)
  MoveL (T19710) to (115.56, 121.34, 20.1) mm, rotated rx 180 ry 0 rz -180 deg; joints [3.351, 66.156, -28.485, 5.473, -37.797, -4.33]
  Call Extruder 0.0456
  MoveL (T19711) to (116.76, 120.14, 20.1) mm, rotated rx 180 ry 0 rz -180 deg; joints [1.409, 65.964, -28.127, 2.297, -37.86, -1.814]
  Call Extruder 0.01356
  MoveL (T19712) to (116.25, 120.14, 20.1) mm, rotated rx 180 ry 0 rz -180 deg; joints [1.407, 66.154, -28.483, 2.302, -37.694, -1.822]
  Call Extruder 0.03951
  MoveL (T19713) to (115.21, 121.18, 20.1) mm, rotated rx 180 ry 0 rz -180 deg; joints [1.407, 66.154, -28.483, 2.302, -37.694, -1.822]
  Call Extruder 0.01356
  MoveL (T19714) to (114.7, 121.18, 20.1) mm, rotated rx 180 ry 0 rz -180 deg; joints [1.365, 65.96, -28.119, 2.225, -37.862, -1.757]
  Call Extruder 0.03951
  MoveL (T19715) to (115.75, 120.14, 20.1) mm, rotated rx 180 ry 0 rz -180 deg; joints [1.365, 65.96, -28.119, 2.225, -37.862, -1.757]
  Call Extruder 0.01356
  MoveL (T19716) to (115.24, 120.14, 20.1) mm, rotated rx 180 ry 0 rz -180 deg; joints [1.365, 65.96, -28.119, 2.225, -37.862, -1.757]
  Call Extruder 0.03951
  MoveL (T19717) to (114.2, 121.18, 20.1) mm, rotated rx 180 ry 0 rz -180 deg; joints [1.365, 65.96, -28.119, 2.225, -37.862, -1.757]
  Call Extruder 0.01356
  MoveL (T19718) to (113.69, 121.18, 20.1) mm, rotated rx 180 ry 0 rz -180 deg; joints [1.365, 65.96, -28.119, 2.225, -37.862, -1.757]
  Call Extruder 0.03951
  MoveL (T19719) to (114.73, 120.14, 20.1) mm, rotated rx 180 ry 0 rz -180 deg; joints [1.319, 71.137, -37.839, 2.402, -33.322, -2.008]
  Call Extruder 0.01356
  MoveL (T19720) to (114.23, 120.14, 20.1) mm, rotated rx 180 ry 0 rz -180 deg; joints [1.319, 71.137, -37.839, 2.402, -33.322, -2.008]
  Call Extruder 0.03951
  MoveL (T19721) to (113.19, 121.18, 20.1) mm, rotated rx 180 ry 0 rz -180 deg; joints [3.282, 71.376, -38.287, 5.995, -33.233, -5.02]
  Call Extruder 0.01356
  MoveL (T19722) to (112.68, 121.18, 20.1) mm, rotated rx 180 ry 0 rz -180 deg; joints [3.282, 71.376, -38.287, 5.995, -33.233, -5.02]
  Call Extruder 0.03951
  MoveL (T19723) to (113.72, 120.14, 20.1) mm, rotated rx 180 ry 0 rz -180 deg; joints [3.398, 66.057, -28.301, 5.538, -37.886, -4.376]
  Call Extruder 0.01356
  MoveL (T19724) to (113.22, 120.14, 20.1) mm, rotated rx 180 ry 0 rz -180 deg; joints [3.398, 66.057, -28.301, 5.538, -37.886, -4.376]
  Call Extruder 0.03951
  MoveL (T19725) to (112.17, 121.18, 20.1) mm, rotated rx 180 ry 0 rz -180 deg; joints [3.398, 66.057, -28.301, 5.538, -37.886, -4.376]
  Call Extruder 0.01356
  MoveL (T19726) to (111.67, 121.18, 20.1) mm, rotated rx 180 ry 0 rz -180 deg; joints [3.398, 66.057, -28.301, 5.538, -37.886, -4.376]
  Call Extruder 0.03951
  MoveL (T19727) to (112.71, 120.14, 20.1) mm, rotated rx 180 ry 0 rz -180 deg; joints [1.366, 65.858, -27.927, 2.222, -37.952, -1.752]
  Call Extruder 0.01356
  MoveL (T19728) to (112.2, 120.14, 20.1) mm, rotated rx 180 ry 0 rz -180 deg; joints [1.366, 65.858, -27.927, 2.222, -37.952, -1.752]
  Call Extruder 0.03951
  MoveL (T19729) to (111.16, 121.18, 20.1) mm, rotated rx 180 ry 0 rz -180 deg; joints [1.366, 65.858, -27.927, 2.222, -37.952, -1.752]
  Call Extruder 0.01356
  MoveL (T19730) to (110.65, 121.18, 20.1) mm, rotated rx 180 ry 0 rz -180 deg; joints [1.366, 65.858, -27.927, 2.222, -37.952, -1.752]
  Call Extruder 0.03951
  MoveL (T19731) to (111.7, 120.14, 20.1) mm, rotated rx 180 ry 0 rz -180 deg; joints [1.365, 65.945, -28.09, 2.224, -37.876, -1.756]
  Call Extruder 0.01356
  MoveL (T19732) to (111.19, 120.14, 20.1) mm, rotated rx 180 ry 0 rz -180 deg; joints [1.365, 65.945, -28.09, 2.224, -37.876, -1.756]
  Call Extruder 0.03951
  MoveL (T19733) to (110.15, 121.18, 20.1) mm, rotated rx 180 ry 0 rz -180 deg; joints [1.365, 65.945, -28.09, 2.224, -37.876, -1.756]
  Call Extruder 0.01356
  MoveL (T19734) to (109.64, 121.18, 20.1) mm, rotated rx 180 ry 0 rz -180 deg; joints [1.365, 65.945, -28.09, 2.224, -37.876, -1.756]
  Call Extruder 0.03951
  MoveL (T19735) to (110.68, 120.14, 20.1) mm, rotated rx 180 ry 0 rz -180 deg; joints [1.365, 65.945, -28.09, 2.224, -37.876, -1.756]
  Call Extruder 0.01356
  MoveL (T19736) to (110.18, 120.14, 20.1) mm, rotated rx 180 ry 0 rz -180 deg; joints [1.365, 65.945, -28.09, 2.224, -37.876, -1.756]
  Call Extruder 0.03951
  MoveL (T19737) to (109.14, 121.18, 20.1) mm, rotated rx 180 ry 0 rz -180 deg; joints [1.332, 65.752, -27.729, 2.162, -38.043, -1.703]
  Call Extruder 0.01356
  MoveL (T19738) to (108.63, 121.18, 20.1) mm, rotated rx 180 ry 0 rz -180 deg; joints [1.332, 65.752, -27.729, 2.162, -38.043, -1.703]
  Call Extruder 0.03951
  MoveL (T19739) to (109.67, 120.14, 20.1) mm, rotated rx 180 ry 0 rz -180 deg; joints [1.332, 65.752, -27.729, 2.162, -38.043, -1.703]
  Call Extruder 0.01356
  MoveL (T19740) to (109.17, 120.14, 20.1) mm, rotated rx 180 ry 0 rz -180 deg; joints [1.332, 65.752, -27.729, 2.162, -38.043, -1.703]
  Call Extruder 0.03951
  MoveL (T19741) to (108.12, 121.18, 20.1) mm, rotated rx 180 ry 0 rz -180 deg; joints [1.323, 65.752, -27.728, 2.147, -38.043, -1.691]
  Call Extruder 0.01356
  MoveL (T19742) to (107.62, 121.18, 20.1) mm, rotated rx 180 ry 0 rz -180 deg; joints [1.323, 65.752, -27.728, 2.147, -38.043, -1.691]
  Call Extruder 0.03951
  MoveL (T19743) to (108.66, 120.14, 20.1) mm, rotated rx 180 ry 0 rz -180 deg; joints [1.276, 71.263, -38.075, 2.33, -33.21, -1.95]
  Call Extruder 0.01356
  MoveL (T19744) to (108.15, 120.14, 20.1) mm, rotated rx 180 ry 0 rz -180 deg; joints [1.276, 71.263, -38.075, 2.33, -33.21, -1.95]
  Call Extruder 0.03951
  MoveL (T19745) to (107.11, 121.18, 20.1) mm, rotated rx 180 ry 0 rz -180 deg; joints [3.322, 71.514, -38.546, 6.088, -33.116, -5.105]
  Call Extruder 0.01356
  MoveL (T19746) to (106.6, 121.18, 20.1) mm, rotated rx 180 ry 0 rz -180 deg; joints [3.322, 71.514, -38.546, 6.088, -33.116, -5.105]
  Call Extruder 0.03951
  MoveL (T19747) to (107.65, 120.14, 20.1) mm, rotated rx 180 ry 0 rz -180 deg; joints [3.322, 71.514, -38.546, 6.088, -33.116, -5.105]
  Call Extruder 0.0016
  MoveL (T19748) to (107.59, 120.14, 20.1) mm, rotated rx 180 ry 0 rz -180 deg; joints [3.445, 65.959, -28.117, 5.603, -37.975, -4.422]
  Call Extruder 0.01196
  MoveL (T19749) to (107.59, 119.69, 20.1) mm, rotated rx 180 ry 0 rz -180 deg; joints [3.445, 65.959, -28.117, 5.603, -37.975, -4.422]
  Call Extruder 0.05642
  MoveL (T19750) to (106.1, 121.18, 20.1) mm, rotated rx 180 ry 0 rz -180 deg; joints [3.445, 65.959, -28.117, 5.603, -37.975, -4.422]
  Call Extruder 0.01356
  MoveL (T19751) to (105.59, 121.18, 20.1) mm, rotated rx 180 ry 0 rz -180 deg; joints [3.445, 65.959, -28.117, 5.603, -37.975, -4.422]
  Call Extruder 0.0756
  MoveL (T19752) to (107.59, 119.19, 20.1) mm, rotated rx 180 ry 0 rz -180 deg; joints [1.339, 65.753, -27.73, 2.173, -38.043, -1.712]
  Call Extruder 0.01356
  MoveL (T19753) to (107.59, 118.68, 20.1) mm, rotated rx 180 ry 0 rz -180 deg; joints [1.339, 65.753, -27.73, 2.173, -38.043, -1.712]
  Call Extruder 0.09478
  MoveL (T19754) to (105.08, 121.18, 20.1) mm, rotated rx 180 ry 0 rz -180 deg; joints [1.339, 65.753, -27.73, 2.173, -38.043, -1.712]
  Call Extruder 0.01356
  MoveL (T19755) to (104.58, 121.18, 20.1) mm, rotated rx 180 ry 0 rz -180 deg; joints [1.339, 65.753, -27.73, 2.173, -38.043, -1.712]
  Call Extruder 0.11396
  MoveL (T19756) to (107.59, 118.17, 20.1) mm, rotated rx 180 ry 0 rz -180 deg; joints [1.326, 65.767, -27.757, 2.152, -38.03, -1.696]
  Call Extruder 0.01356
  MoveL (T19757) to (107.59, 117.67, 20.1) mm, rotated rx 180 ry 0 rz -180 deg; joints [1.326, 65.767, -27.757, 2.152, -38.03, -1.696]
  Call Extruder 0.13313
  MoveL (T19758) to (104.07, 121.18, 20.1) mm, rotated rx 180 ry 0 rz -180 deg; joints [1.326, 65.767, -27.757, 2.152, -38.03, -1.696]
  Call Extruder 0.00678
  MoveL (T19759) to (103.82, 121.18, 20.1) mm, rotated rx 180 ry 0 rz -180 deg; joints [1.326, 65.767, -27.757, 2.152, -38.03, -1.696]
  Call Extruder 0.00678
  MoveL (T19760) to (103.82, 120.93, 20.1) mm, rotated rx 180 ry 0 rz -180 deg; joints [1.326, 65.767, -27.757, 2.152, -38.03, -1.696]
  Call Extruder 0.14272
  MoveL (T19761) to (107.59, 117.16, 20.1) mm, rotated rx 180 ry 0 rz -180 deg; joints [1.326, 65.767, -27.757, 2.152, -38.03, -1.696]
  Call Extruder 0.01356
  MoveL (T19762) to (107.59, 116.65, 20.1) mm, rotated rx 180 ry 0 rz -180 deg; joints [1.326, 65.767, -27.757, 2.152, -38.03, -1.696]
  Call Extruder 0.14272
  MoveL (T19763) to (103.82, 120.42, 20.1) mm, rotated rx 180 ry 0 rz -180 deg; joints [1.326, 65.767, -27.757, 2.152, -38.03, -1.696]
  Call Extruder 0.01356
  MoveL (T19764) to (103.82, 119.92, 20.1) mm, rotated rx 180 ry 0 rz -180 deg; joints [1.326, 65.767, -27.757, 2.152, -38.03, -1.696]
  Call Extruder 0.25455
  MoveL (T19765) to (110.54, 113.2, 20.1) mm, rotated rx 180 ry 0 rz -180 deg; joints [1.326, 65.767, -27.757, 2.152, -38.03, -1.696]
  Call Extruder 0.01008
  MoveL (T19766) to (110.37, 112.86, 20.1) mm, rotated rx 180 ry 0 rz -180 deg; joints [1.323, 65.752, -27.728, 2.147, -38.043, -1.691]
  Call Extruder 0.24807
  MoveL (T19767) to (103.82, 119.41, 20.1) mm, rotated rx 180 ry 0 rz -180 deg; joints [1.323, 65.752, -27.728, 2.147, -38.043, -1.691]
  Call Extruder 0.01356
  MoveL (T19768) to (103.82, 118.9, 20.1) mm, rotated rx 180 ry 0 rz -180 deg; joints [1.323, 65.752, -27.728, 2.147, -38.043, -1.691]
  Call Extruder 0.24159
  MoveL (T19769) to (110.2, 112.53, 20.1) mm, rotated rx 180 ry 0 rz -180 deg; joints [1.321, 65.987, -28.169, 2.154, -37.837, -1.701]
  Call Extruder 0.01008
  MoveL (T19770) to (110.03, 112.19, 20.1) mm, rotated rx 180 ry 0 rz -180 deg; joints [1.321, 65.987, -28.169, 2.154, -37.837, -1.701]
  Call Extruder 0.23512
  MoveL (T19771) to (103.82, 118.4, 20.1) mm, rotated rx 180 ry 0 rz -180 deg; joints [1.321, 65.987, -28.169, 2.154, -37.837, -1.701]
  Call Extruder 0.01356
  MoveL (T19772) to (103.82, 117.89, 20.1) mm, rotated rx 180 ry 0 rz -180 deg; joints [1.321, 65.987, -28.169, 2.154, -37.837, -1.701]
  Call Extruder 0.22864
  MoveL (T19773) to (109.86, 111.86, 20.1) mm, rotated rx 180 ry 0 rz -180 deg; joints [1.321, 65.987, -28.169, 2.154, -37.837, -1.701]
  Call Extruder 0.01008
  MoveL (T19774) to (109.68, 111.52, 20.1) mm, rotated rx 180 ry 0 rz -180 deg; joints [1.321, 65.987, -28.169, 2.154, -37.837, -1.701]
  Call Extruder 0.22216
  MoveL (T19775) to (103.82, 117.38, 20.1) mm, rotated rx 180 ry 0 rz -180 deg; joints [1.321, 65.987, -28.169, 2.154, -37.837, -1.701]
  Call Extruder 0.01356
  MoveL (T19776) to (103.82, 116.88, 20.1) mm, rotated rx 180 ry 0 rz -180 deg; joints [1.321, 65.987, -28.169, 2.154, -37.837, -1.701]
  Call Extruder 0.21568
  MoveL (T19777) to (109.51, 111.18, 20.1) mm, rotated rx 180 ry 0 rz -180 deg; joints [1.321, 65.987, -28.169, 2.154, -37.837, -1.701]
  Call Extruder 0.01008
  MoveL (T19778) to (109.34, 110.85, 20.1) mm, rotated rx 180 ry 0 rz -180 deg; joints [1.707, 65.826, -28.275, 2.799, -37.585, -2.218]
  Call Extruder 0.2092
  MoveL (T19779) to (103.82, 116.37, 20.1) mm, rotated rx 180 ry 0 rz -180 deg; joints [1.707, 65.826, -28.275, 2.799, -37.585, -2.218]
  Call Extruder 0.01356
  MoveL (T19780) to (103.82, 115.86, 20.1) mm, rotated rx 180 ry 0 rz -180 deg; joints [1.707, 66.062, -28.309, 2.786, -37.785, -2.202]
  Call Extruder 0.20272
  MoveL (T19781) to (109.17, 110.51, 20.1) mm, rotated rx 180 ry 0 rz -180 deg; joints [1.707, 66.062, -28.309, 2.786, -37.785, -2.202]
  Call Extruder 0.01008
  MoveL (T19782) to (109, 110.18, 20.1) mm, rotated rx 180 ry 0 rz -180 deg; joints [1.707, 66.062, -28.309, 2.786, -37.785, -2.202]
  Call Extruder 0.19624
  MoveL (T19783) to (103.82, 115.36, 20.1) mm, rotated rx 180 ry 0 rz -180 deg; joints [1.707, 66.062, -28.309, 2.786, -37.785, -2.202]
  Call Extruder 0.01356
  MoveL (T19784) to (103.82, 114.85, 20.1) mm, rotated rx 180 ry 0 rz -180 deg; joints [1.707, 66.062, -28.309, 2.786, -37.785, -2.202]
  Call Extruder 0.18977
  MoveL (T19785) to (108.83, 109.84, 20.1) mm, rotated rx 180 ry 0 rz -180 deg; joints [1.707, 66.062, -28.309, 2.786, -37.785, -2.202]
  Call Extruder 0.01008
  MoveL (T19786) to (108.66, 109.51, 20.1) mm, rotated rx 180 ry 0 rz -180 deg; joints [1.707, 66.062, -28.309, 2.786, -37.785, -2.202]
  Call Extruder 0.18329
  MoveL (T19787) to (103.82, 114.35, 20.1) mm, rotated rx 180 ry 0 rz -180 deg; joints [1.707, 66.062, -28.309, 2.786, -37.785, -2.202]
  Call Extruder 0.01356
  MoveL (T19788) to (103.82, 113.84, 20.1) mm, rotated rx 180 ry 0 rz -180 deg; joints [1.707, 66.062, -28.309, 2.786, -37.785, -2.202]
  Call Extruder 0.17681
  MoveL (T19789) to (108.49, 109.17, 20.1) mm, rotated rx 180 ry 0 rz -180 deg; joints [1.707, 66.062, -28.309, 2.786, -37.785, -2.202]
  Call Extruder 0.01008
  MoveL (T19790) to (108.32, 108.84, 20.1) mm, rotated rx 180 ry 0 rz -180 deg; joints [1.707, 66.062, -28.309, 2.786, -37.785, -2.202]
  Call Extruder 0.17033
  MoveL (T19791) to (103.82, 113.33, 20.1) mm, rotated rx 180 ry 0 rz -180 deg; joints [1.442, 66.044, -28.277, 2.353, -37.791, -1.86]
  Call Extruder 0.01356
  MoveL (T19792) to (103.82, 112.83, 20.1) mm, rotated rx 180 ry 0 rz -180 deg; joints [1.442, 66.044, -28.277, 2.353, -37.791, -1.86]
  Call Extruder 0.16385
  MoveL (T19793) to (108.14, 108.5, 20.1) mm, rotated rx 180 ry 0 rz -180 deg; joints [1.442, 66.044, -28.277, 2.353, -37.791, -1.86]
  Call Extruder 0.01008
  MoveL (T19794) to (107.97, 108.17, 20.1) mm, rotated rx 180 ry 0 rz -180 deg; joints [1.657, 66.06, -28.305, 2.705, -37.785, -2.139]
  Call Extruder 0.15737
  MoveL (T19795) to (103.82, 112.32, 20.1) mm, rotated rx 180 ry 0 rz -180 deg; joints [1.657, 66.06, -28.305, 2.705, -37.785, -2.139]
  Call Extruder 0.01356
  MoveL (T19796) to (103.82, 111.81, 20.1) mm, rotated rx 180 ry 0 rz -180 deg; joints [1.657, 66.06, -28.305, 2.705, -37.785, -2.139]
  Call Extruder 0.1509
  MoveL (T19797) to (107.8, 107.83, 20.1) mm, rotated rx 180 ry 0 rz -180 deg; joints [1.679, 66.082, -28.348, 2.742, -37.766, -2.168]
  Call Extruder 0.01008
  MoveL (T19798) to (107.63, 107.5, 20.1) mm, rotated rx 180 ry 0 rz -180 deg; joints [1.679, 66.082, -28.348, 2.742, -37.766, -2.168]
  Call Extruder 0.14442
  MoveL (T19799) to (103.82, 111.31, 20.1) mm, rotated rx 180 ry 0 rz -180 deg; joints [1.743, 66.244, -28.651, 2.855, -37.627, -2.262]
  Call Extruder 0.01356
  MoveL (T19800) to (103.82, 110.8, 20.1) mm, rotated rx 180 ry 0 rz -180 deg; joints [1.743, 66.244, -28.651, 2.855, -37.627, -2.262]
  Call Extruder 0.13954
  MoveL (T19801) to (107.5, 107.12, 20.1) mm, rotated rx 180 ry 0 rz -180 deg; joints [1.743, 66.244, -28.651, 2.855, -37.627, -2.262]
  Call Extruder 0.01356
  MoveL (T19802) to (107.5, 106.61, 20.1) mm, rotated rx 180 ry 0 rz -180 deg; joints [1.821, 66.07, -28.325, 2.972, -37.782, -2.35]
  Call Extruder 0.13954
  MoveL (T19803) to (103.82, 110.3, 20.1) mm, rotated rx 180 ry 0 rz -180 deg; joints [1.821, 66.07, -28.325, 2.972, -37.782, -2.35]
  Call Extruder 0.01356
  MoveL (T19804) to (103.82, 109.79, 20.1) mm, rotated rx 180 ry 0 rz -180 deg; joints [1.821, 66.07, -28.325, 2.972, -37.782, -2.35]
  Call Extruder 0.14563
  MoveL (T19805) to (107.66, 105.95, 20.1) mm, rotated rx 180 ry 0 rz -180 deg; joints [1.821, 66.07, -28.325, 2.972, -37.782, -2.35]
  Set speed (45.0 mm/s)
  Call Extruder -1.6
  MoveL (T19806) to (107.66, 105.95, 20.1) mm, rotated rx 180 ry 0 rz -180 deg; joints [1.821, 66.07, -28.325, 2.972, -37.782, -2.35]
  Set speed (120.0 mm/s)
  MoveL (T19807) to (107.66, 105.95, 20.1) mm, rotated rx 180 ry 0 rz -180 deg; joints [1.941, 66.079, -28.342, 3.169, -37.779, -2.506]
  Call Extruder -0.38
  MoveL (T19808) to (106.91, 106.7, 20.1) mm, rotated rx 180 ry 0 rz -180 deg; joints [3.239, 69.732, -35.198, 5.7, -34.666, -4.693]
  Set speed (45.0 mm/s)
  Call Extruder -0.02
  MoveL (T19809) to (106.91, 106.7, 20.1) mm, rotated rx 180 ry 0 rz -180 deg; joints [3.239, 69.732, -35.198, 5.7, -34.666, -4.693]
  Set speed (150.0 mm/s)
  MoveL (T19810) to (106.91, 106.7, 22.1) mm, rotated rx 180 ry 0 rz -180 deg; joints [3.232, 70.063, -35.82, 5.731, -34.376, -4.735]
  MoveL (T19811) to (109.44, 103.66, 22.1) mm, rotated rx 180 ry 0 rz -180 deg; joints [3.232, 70.063, -35.82, 5.731, -34.376, -4.735]
  MoveL (T19812) to (109.44, 103.66, 20.1) mm, rotated rx 180 ry 0 rz -180 deg; joints [3.232, 70.063, -35.82, 5.731, -34.376, -4.735]
  Set speed (40.0 mm/s)
  Call Extruder 2.0
  MoveL (T19813) to (109.44, 103.66, 20.1) mm, rotated rx 180 ry 0 rz -180 deg; joints [2.845, 71.079, -37.73, 5.166, -33.457, -4.313]
  Set speed (25.0 mm/s)
  MoveL (T19814) to (109.44, 103.66, 20.1) mm, rotated rx 180 ry 0 rz -180 deg; joints [2.845, 71.079, -37.73, 5.166, -33.457, -4.313]
  Call Extruder 0.05792
  MoveL (T19815) to (107.92, 105.19, 20.1) mm, rotated rx 180 ry 0 rz -180 deg; joints [3.211, 71.138, -37.839, 5.835, -33.435, -4.875]
  Call Extruder 0.01107
  MoveL (T19816) to (107.5, 105.19, 20.1) mm, rotated rx 180 ry 0 rz -180 deg; joints [3.211, 71.138, -37.839, 5.835, -33.435, -4.875]
  Call Extruder 0.01107
  MoveL (T19817) to (107.5, 105.6, 20.1) mm, rotated rx 180 ry 0 rz -180 deg; joints [3.211, 71.138, -37.839, 5.835, -33.435, -4.875]
  Call Extruder 0.13954
  MoveL (T19818) to (103.82, 109.28, 20.1) mm, rotated rx 180 ry 0 rz -180 deg; joints [1.893, 67.206, -30.457, 3.162, -36.791, -2.533]
  Call Extruder 0.01356
  MoveL (T19819) to (103.82, 108.78, 20.1) mm, rotated rx 180 ry 0 rz -180 deg; joints [1.893, 67.206, -30.457, 3.162, -36.791, -2.533]
  Call Extruder 0.18784
  MoveL (T19820) to (108.78, 103.82, 20.1) mm, rotated rx 180 ry 0 rz -180 deg; joints [1.893, 67.206, -30.457, 3.162, -36.791, -2.533]
  Call Extruder 0.01356
  MoveL (T19821) to (108.27, 103.82, 20.1) mm, rotated rx 180 ry 0 rz -180 deg; joints [1.895, 67.069, -30.2, 3.156, -36.911, -2.524]
  Call Extruder 0.16866
  MoveL (T19822) to (103.82, 108.27, 20.1) mm, rotated rx 180 ry 0 rz -180 deg; joints [1.895, 67.069, -30.2, 3.156, -36.911, -2.524]
  Call Extruder 0.01356
  MoveL (T19823) to (103.82, 107.77, 20.1) mm, rotated rx 180 ry 0 rz -180 deg; joints [1.895, 67.069, -30.2, 3.156, -36.911, -2.524]
  Call Extruder 0.14948
  MoveL (T19824) to (107.77, 103.82, 20.1) mm, rotated rx 180 ry 0 rz -180 deg; joints [2.319, 66.113, -28.405, 3.789, -37.768, -2.997]
  Call Extruder 0.01356
  MoveL (T19825) to (107.26, 103.82, 20.1) mm, rotated rx 180 ry 0 rz -180 deg; joints [2.319, 66.113, -28.405, 3.789, -37.768, -2.997]
  Call Extruder 0.13031
  MoveL (T19826) to (103.82, 107.26, 20.1) mm, rotated rx 180 ry 0 rz -180 deg; joints [2.319, 66.113, -28.405, 3.789, -37.768, -2.997]
  Call Extruder 0.01356
  MoveL (T19827) to (103.82, 106.75, 20.1) mm, rotated rx 180 ry 0 rz -180 deg; joints [2.44, 66.125, -28.427, 3.986, -37.764, -3.153]
  Call Extruder 0.11113
  MoveL (T19828) to (106.75, 103.82, 20.1) mm, rotated rx 180 ry 0 rz -180 deg; joints [2.44, 66.125, -28.427, 3.986, -37.764, -3.153]
  Call Extruder 0.01356
  MoveL (T19829) to (106.25, 103.82, 20.1) mm, rotated rx 180 ry 0 rz -180 deg; joints [2.44, 66.125, -28.427, 3.986, -37.764, -3.153]
  Call Extruder 0.09195
  MoveL (T19830) to (103.82, 106.25, 20.1) mm, rotated rx 180 ry 0 rz -180 deg; joints [2.44, 66.125, -28.427, 3.986, -37.764, -3.153]
  Call Extruder 0.01356
  MoveL (T19831) to (103.82, 105.74, 20.1) mm, rotated rx 180 ry 0 rz -180 deg; joints [3.266, 68.405, -32.708, 5.586, -35.827, -4.534]
  Call Extruder 0.07277
  MoveL (T19832) to (105.74, 103.82, 20.1) mm, rotated rx 180 ry 0 rz -180 deg; joints [3.266, 68.405, -32.708, 5.586, -35.827, -4.534]
  Call Extruder 0.01356
  MoveL (T19833) to (105.23, 103.82, 20.1) mm, rotated rx 180 ry 0 rz -180 deg; joints [3.266, 68.405, -32.708, 5.586, -35.827, -4.534]
  Call Extruder 0.05359
  MoveL (T19834) to (103.82, 105.23, 20.1) mm, rotated rx 180 ry 0 rz -180 deg; joints [3.26, 68.719, -33.297, 5.612, -35.552, -4.571]
  Call Extruder 0.01356
  MoveL (T19835) to (103.82, 104.73, 20.1) mm, rotated rx 180 ry 0 rz -180 deg; joints [3.26, 68.719, -33.297, 5.612, -35.552, -4.571]
  Call Extruder 0.03442
  MoveL (T19836) to (104.73, 103.82, 20.1) mm, rotated rx 180 ry 0 rz -180 deg; joints [2.685, 70.151, -35.986, 4.773, -34.258, -3.948]
  Call Extruder 0.01356
  MoveL (T19837) to (104.22, 103.82, 20.1) mm, rotated rx 180 ry 0 rz -180 deg; joints [2.685, 70.151, -35.986, 4.773, -34.258, -3.948]
  Call Extruder 0.02132
  MoveL (T19838) to (103.66, 104.38, 20.1) mm, rotated rx 180 ry 0 rz -180 deg; joints [2.685, 70.151, -35.986, 4.773, -34.258, -3.948]
  Set speed (45.0 mm/s)
  Call Extruder -1.6
  MoveL (T19839) to (103.66, 104.38, 20.1) mm, rotated rx 180 ry 0 rz -180 deg; joints [2.754, 70.37, -36.398, 4.92, -34.07, -4.079]
  Set speed (120.0 mm/s)
  MoveL (T19840) to (103.66, 104.38, 20.1) mm, rotated rx 180 ry 0 rz -180 deg; joints [2.754, 70.37, -36.398, 4.92, -34.07, -4.079]
  Call Extruder -0.28359
  MoveL (T19841) to (104.22, 103.82, 20.1) mm, rotated rx 180 ry 0 rz -180 deg; joints [2.754, 70.37, -36.398, 4.92, -34.07, -4.079]
  Call Extruder -0.09641
  MoveL (T19842) to (104.49, 103.82, 20.1) mm, rotated rx 180 ry 0 rz -180 deg; joints [2.762, 70.433, -36.516, 4.941, -34.016, -4.099]
  Set speed (45.0 mm/s)
  Call Extruder -0.02
  MoveL (T19843) to (104.49, 103.82, 20.1) mm, rotated rx 180 ry 0 rz -180 deg; joints [2.756, 70.817, -37.236, 4.973, -33.68, -4.142]
  Set speed (150.0 mm/s)
  MoveL (T19844) to (104.49, 103.82, 22.1) mm, rotated rx 180 ry 0 rz -180 deg; joints [2.756, 70.817, -37.236, 4.973, -33.68, -4.142]
  MoveL (T19845) to (102.7, 122.25, 22.1) mm, rotated rx 180 ry 0 rz -180 deg; joints [2.756, 70.817, -37.236, 4.973, -33.68, -4.142]
  MoveL (T19846) to (102.7, 122.25, 20.1) mm, rotated rx 180 ry 0 rz -180 deg; joints [2.756, 70.817, -37.236, 4.973, -33.68, -4.142]
  Set speed (40.0 mm/s)
  Call Extruder 2.0
  MoveL (T19847) to (102.7, 122.25, 20.1) mm, rotated rx 180 ry 0 rz -180 deg; joints [2.756, 70.817, -37.236, 4.973, -33.68, -4.142]
  Set speed (15.0 mm/s)
  MoveL (T19848) to (102.7, 122.25, 20.1) mm, rotated rx 180 ry 0 rz -180 deg; joints [2.756, 70.817, -37.236, 4.973, -33.68, -4.142]
  Call Extruder 0.02194
  MoveL (T19849) to (122.25, 122.25, 20.1) mm, rotated rx 180 ry 0 rz -180 deg; joints [2.756, 70.817, -37.236, 4.973, -33.68, -4.142]
  Call Extruder 0.00011
  MoveL (T19850) to (122.25, 122.15, 20.1) mm, rotated rx 180 ry 0 rz -180 deg; joints [2.756, 70.817, -37.236, 4.973, -33.68, -4.142]
  Call Extruder 0.02189
  MoveL (T19851) to (102.75, 122.15, 20.1) mm, rotated rx 180 ry 0 rz -180 deg; joints [2.756, 70.817, -37.236, 4.973, -33.68, -4.142]
  Call Extruder 0.00011
  MoveL (T19852) to (102.75, 122.05, 20.1) mm, rotated rx 180 ry 0 rz -180 deg; joints [2.756, 70.817, -37.236, 4.973, -33.68, -4.142]
  Call Extruder 0.02189
  MoveL (T19853) to (122.25, 122.05, 20.1) mm, rotated rx 180 ry 0 rz -180 deg; joints [2.756, 70.817, -37.236, 4.973, -33.68, -4.142]
  Call Extruder 0.00011
  MoveL (T19854) to (122.25, 121.95, 20.1) mm, rotated rx 180 ry 0 rz -180 deg; joints [2.756, 70.817, -37.236, 4.973, -33.68, -4.142]
  Call Extruder 0.02189
  MoveL (T19855) to (102.75, 121.95, 20.1) mm, rotated rx 180 ry 0 rz -180 deg; joints [2.761, 70.488, -36.618, 4.946, -33.968, -4.105]
  Call Extruder 0.00011
  MoveL (T19856) to (102.75, 121.85, 20.1) mm, rotated rx 180 ry 0 rz -180 deg; joints [2.761, 70.488, -36.618, 4.946, -33.968, -4.105]
  Call Extruder 0.02189
  MoveL (T19857) to (122.25, 121.85, 20.1) mm, rotated rx 180 ry 0 rz -180 deg; joints [2.761, 70.488, -36.618, 4.946, -33.968, -4.105]
  Call Extruder 0.00011
  MoveL (T19858) to (122.25, 121.75, 20.1) mm, rotated rx 180 ry 0 rz -180 deg; joints [2.761, 70.488, -36.618, 4.946, -33.968, -4.105]
  Call Extruder 0.02189
  MoveL (T19859) to (102.75, 121.75, 20.1) mm, rotated rx 180 ry 0 rz -180 deg; joints [2.761, 70.488, -36.618, 4.946, -33.968, -4.105]
  Call Extruder 0.00011
  MoveL (T19860) to (102.75, 121.65, 20.1) mm, rotated rx 180 ry 0 rz -180 deg; joints [2.761, 70.488, -36.618, 4.946, -33.968, -4.105]
  Call Extruder 0.02189
  MoveL (T19861) to (122.25, 121.65, 20.1) mm, rotated rx 180 ry 0 rz -180 deg; joints [2.761, 70.488, -36.618, 4.946, -33.968, -4.105]
  Call Extruder 0.00011
  MoveL (T19862) to (122.25, 121.55, 20.1) mm, rotated rx 180 ry 0 rz -180 deg; joints [2.761, 70.256, -36.578, 4.97, -33.777, -4.135]
  Call Extruder 0.02189
  MoveL (T19863) to (102.75, 121.55, 20.1) mm, rotated rx 180 ry 0 rz -180 deg; joints [1.813, 70.499, -37.034, 3.285, -33.508, -2.74]
  Call Extruder 0.00011
  MoveL (T19864) to (102.75, 121.45, 20.1) mm, rotated rx 180 ry 0 rz -180 deg; joints [1.813, 70.73, -37.074, 3.269, -33.699, -2.72]
  Call Extruder 0.02189
  MoveL (T19865) to (122.25, 121.45, 20.1) mm, rotated rx 180 ry 0 rz -180 deg; joints [1.813, 70.73, -37.074, 3.269, -33.699, -2.72]
  Call Extruder 0.00011
  MoveL (T19866) to (122.25, 121.35, 20.1) mm, rotated rx 180 ry 0 rz -180 deg; joints [1.813, 70.73, -37.074, 3.269, -33.699, -2.72]
  Call Extruder 0.02189
  MoveL (T19867) to (102.75, 121.35, 20.1) mm, rotated rx 180 ry 0 rz -180 deg; joints [1.813, 70.73, -37.074, 3.269, -33.699, -2.72]
  Call Extruder 0.00011
  MoveL (T19868) to (102.75, 121.25, 20.1) mm, rotated rx 180 ry 0 rz -180 deg; joints [1.813, 70.73, -37.074, 3.269, -33.699, -2.72]
  Call Extruder 0.02189
  MoveL (T19869) to (122.25, 121.25, 20.1) mm, rotated rx 180 ry 0 rz -180 deg; joints [1.813, 70.73, -37.074, 3.269, -33.699, -2.72]
  Call Extruder 0.00011
  MoveL (T19870) to (122.25, 121.15, 20.1) mm, rotated rx 180 ry 0 rz -180 deg; joints [1.813, 70.73, -37.074, 3.269, -33.699, -2.72]
  Call Extruder 0.02189
  MoveL (T19871) to (102.75, 121.15, 20.1) mm, rotated rx 180 ry 0 rz -180 deg; joints [1.813, 70.73, -37.074, 3.269, -33.699, -2.72]
  Call Extruder 0.00011
  MoveL (T19872) to (102.75, 121.05, 20.1) mm, rotated rx 180 ry 0 rz -180 deg; joints [1.813, 70.73, -37.074, 3.269, -33.699, -2.72]
  Call Extruder 0.02189
  MoveL (T19873) to (122.25, 121.05, 20.1) mm, rotated rx 180 ry 0 rz -180 deg; joints [1.886, 70.961, -37.507, 3.418, -33.501, -2.851]
  Call Extruder 0.00011
  MoveL (T19874) to (122.25, 120.95, 20.1) mm, rotated rx 180 ry 0 rz -180 deg; joints [1.886, 70.961, -37.507, 3.418, -33.501, -2.851]
  Call Extruder 0.02189
  MoveL (T19875) to (102.75, 120.95, 20.1) mm, rotated rx 180 ry 0 rz -180 deg; joints [1.886, 70.961, -37.507, 3.418, -33.501, -2.851]
  Call Extruder 0.00011
  MoveL (T19876) to (102.75, 120.85, 20.1) mm, rotated rx 180 ry 0 rz -180 deg; joints [1.946, 70.967, -37.519, 3.528, -33.498, -2.943]
  Call Extruder 0.02189
  MoveL (T19877) to (122.25, 120.85, 20.1) mm, rotated rx 180 ry 0 rz -180 deg; joints [1.946, 70.967, -37.519, 3.528, -33.498, -2.943]
  Call Extruder 0.00011
  MoveL (T19878) to (122.25, 120.75, 20.1) mm, rotated rx 180 ry 0 rz -180 deg; joints [1.833, 70.61, -36.848, 3.296, -33.806, -2.74]
  Call Extruder 0.02189
  MoveL (T19879) to (102.75, 120.75, 20.1) mm, rotated rx 180 ry 0 rz -180 deg; joints [1.833, 70.61, -36.848, 3.296, -33.806, -2.74]
  Call Extruder 0.00011
  MoveL (T19880) to (102.75, 120.65, 20.1) mm, rotated rx 180 ry 0 rz -180 deg; joints [1.833, 70.61, -36.848, 3.296, -33.806, -2.74]
  Call Extruder 0.02189
  MoveL (T19881) to (122.25, 120.65, 20.1) mm, rotated rx 180 ry 0 rz -180 deg; joints [1.835, 70.432, -36.514, 3.286, -33.962, -2.727]
  Call Extruder 0.00011
  MoveL (T19882) to (122.25, 120.55, 20.1) mm, rotated rx 180 ry 0 rz -180 deg; joints [1.835, 70.432, -36.514, 3.286, -33.962, -2.727]
  Call Extruder 0.02189
  MoveL (T19883) to (102.75, 120.55, 20.1) mm, rotated rx 180 ry 0 rz -180 deg; joints [1.835, 70.432, -36.514, 3.286, -33.962, -2.727]
  Call Extruder 0.00011
  MoveL (T19884) to (102.75, 120.45, 20.1) mm, rotated rx 180 ry 0 rz -180 deg; joints [2.007, 70.973, -37.53, 3.638, -33.496, -3.035]
  Call Extruder 0.02189
  MoveL (T19885) to (122.25, 120.45, 20.1) mm, rotated rx 180 ry 0 rz -180 deg; joints [2.007, 70.973, -37.53, 3.638, -33.496, -3.035]
  Call Extruder 0.00011
  MoveL (T19886) to (122.25, 120.35, 20.1) mm, rotated rx 180 ry 0 rz -180 deg; joints [2.007, 70.973, -37.53, 3.638, -33.496, -3.035]
  Call Extruder 0.02189
  MoveL (T19887) to (102.75, 120.35, 20.1) mm, rotated rx 180 ry 0 rz -180 deg; joints [2.068, 70.98, -37.542, 3.749, -33.494, -3.128]
  Call Extruder 0.00011
  MoveL (T19888) to (102.75, 120.25, 20.1) mm, rotated rx 180 ry 0 rz -180 deg; joints [2.068, 70.98, -37.542, 3.749, -33.494, -3.128]
  Call Extruder 0.02189
  MoveL (T19889) to (122.25, 120.25, 20.1) mm, rotated rx 180 ry 0 rz -180 deg; joints [2.068, 70.98, -37.542, 3.749, -33.494, -3.128]
  Call Extruder 0.00011
  MoveL (T19890) to (122.25, 120.15, 20.1) mm, rotated rx 180 ry 0 rz -180 deg; joints [1.852, 70.3, -36.266, 3.306, -34.078, -2.739]
  Call Extruder 0.02189
  MoveL (T19891) to (102.75, 120.15, 20.1) mm, rotated rx 180 ry 0 rz -180 deg; joints [1.852, 70.3, -36.266, 3.306, -34.078, -2.739]
  Call Extruder 0.00011
  MoveL (T19892) to (102.75, 120.05, 20.1) mm, rotated rx 180 ry 0 rz -180 deg; joints [1.852, 70.3, -36.266, 3.306, -34.078, -2.739]
  Call Extruder 0.02189
  MoveL (T19893) to (122.25, 120.05, 20.1) mm, rotated rx 180 ry 0 rz -180 deg; joints [1.883, 70.216, -36.107, 3.355, -34.154, -2.778]
  Call Extruder 0.00011
  MoveL (T19894) to (122.25, 119.95, 20.1) mm, rotated rx 180 ry 0 rz -180 deg; joints [1.883, 70.216, -36.107, 3.355, -34.154, -2.778]
  Call Extruder 0.02189
  MoveL (T19895) to (102.75, 119.95, 20.1) mm, rotated rx 180 ry 0 rz -180 deg; joints [1.883, 70.216, -36.107, 3.355, -34.154, -2.778]
  Call Extruder 0.00011
  MoveL (T19896) to (102.75, 119.85, 20.1) mm, rotated rx 180 ry 0 rz -180 deg; joints [1.883, 70.216, -36.107, 3.355, -34.154, -2.778]
  Call Extruder 0.02189
  MoveL (T19897) to (122.25, 119.85, 20.1) mm, rotated rx 180 ry 0 rz -180 deg; joints [2.129, 70.986, -37.555, 3.859, -33.491, -3.22]
  Call Extruder 0.00011
  MoveL (T19898) to (122.25, 119.75, 20.1) mm, rotated rx 180 ry 0 rz -180 deg; joints [2.129, 70.986, -37.555, 3.859, -33.491, -3.22]
  Call Extruder 0.02189
  MoveL (T19899) to (102.75, 119.75, 20.1) mm, rotated rx 180 ry 0 rz -180 deg; joints [2.129, 70.986, -37.555, 3.859, -33.491, -3.22]
  Call Extruder 0.00011
  MoveL (T19900) to (102.75, 119.65, 20.1) mm, rotated rx 180 ry 0 rz -180 deg; joints [2.189, 70.993, -37.568, 3.97, -33.489, -3.312]
  Call Extruder 0.02189
  MoveL (T19901) to (122.25, 119.65, 20.1) mm, rotated rx 180 ry 0 rz -180 deg; joints [2.189, 70.993, -37.568, 3.97, -33.489, -3.312]
  Call Extruder 0.00011
  MoveL (T19902) to (122.25, 119.55, 20.1) mm, rotated rx 180 ry 0 rz -180 deg; joints [1.915, 70.131, -35.948, 3.405, -34.23, -2.816]
  Call Extruder 0.02189
  MoveL (T19903) to (102.75, 119.55, 20.1) mm, rotated rx 180 ry 0 rz -180 deg; joints [1.915, 70.131, -35.948, 3.405, -34.23, -2.816]
  Call Extruder 0.00011
  MoveL (T19904) to (102.75, 119.45, 20.1) mm, rotated rx 180 ry 0 rz -180 deg; joints [1.915, 70.131, -35.948, 3.405, -34.23, -2.816]
  Call Extruder 0.02189
  MoveL (T19905) to (122.25, 119.45, 20.1) mm, rotated rx 180 ry 0 rz -180 deg; joints [1.946, 70.046, -35.79, 3.455, -34.305, -2.855]
  Call Extruder 0.00011
  MoveL (T19906) to (122.25, 119.35, 20.1) mm, rotated rx 180 ry 0 rz -180 deg; joints [1.946, 70.046, -35.79, 3.455, -34.305, -2.855]
  Call Extruder 0.02189
  MoveL (T19907) to (102.75, 119.35, 20.1) mm, rotated rx 180 ry 0 rz -180 deg; joints [2.25, 71, -37.581, 4.08, -33.486, -3.405]
  Call Extruder 0.00011
  MoveL (T19908) to (102.75, 119.25, 20.1) mm, rotated rx 180 ry 0 rz -180 deg; joints [2.311, 71.007, -37.595, 4.191, -33.483, -3.497]
  Call Extruder 0.02189
  MoveL (T19909) to (122.25, 119.25, 20.1) mm, rotated rx 180 ry 0 rz -180 deg; joints [2.311, 71.007, -37.595, 4.191, -33.483, -3.497]
  Call Extruder 0.00011
  MoveL (T19910) to (122.25, 119.15, 20.1) mm, rotated rx 180 ry 0 rz -180 deg; joints [2.311, 71.007, -37.595, 4.191, -33.483, -3.497]
  Call Extruder 0.02189
  MoveL (T19911) to (102.75, 119.15, 20.1) mm, rotated rx 180 ry 0 rz -180 deg; joints [1.978, 69.963, -35.633, 3.504, -34.38, -2.893]
  Call Extruder 0.00011
  MoveL (T19912) to (102.75, 119.05, 20.1) mm, rotated rx 180 ry 0 rz -180 deg; joints [1.978, 69.963, -35.633, 3.504, -34.38, -2.893]
  Call Extruder 0.02189
  MoveL (T19913) to (122.25, 119.05, 20.1) mm, rotated rx 180 ry 0 rz -180 deg; joints [1.978, 69.963, -35.633, 3.504, -34.38, -2.893]
  Call Extruder 0.00011
  MoveL (T19914) to (122.25, 118.95, 20.1) mm, rotated rx 180 ry 0 rz -180 deg; joints [1.978, 69.963, -35.633, 3.504, -34.38, -2.893]
  Call Extruder 0.00626
  MoveL (T19915) to (116.68, 118.95, 20.1) mm, rotated rx 180 ry 0 rz -180 deg; joints [2.009, 69.879, -35.475, 3.553, -34.455, -2.931]
  Call Extruder 0.00011
  MoveL (T19916) to (116.68, 118.85, 20.1) mm, rotated rx 180 ry 0 rz -180 deg; joints [2.009, 69.879, -35.475, 3.553, -34.455, -2.931]
  Call Extruder 0.00626
  MoveL (T19917) to (122.25, 118.85, 20.1) mm, rotated rx 180 ry 0 rz -180 deg; joints [2.009, 69.879, -35.475, 3.553, -34.455, -2.931]
  Call Extruder 0.00011
  MoveL (T19918) to (122.25, 118.75, 20.1) mm, rotated rx 180 ry 0 rz -180 deg; joints [2.371, 71.015, -37.608, 4.302, -33.481, -3.59]
  Call Extruder 0.00626
  MoveL (T19919) to (116.68, 118.75, 20.1) mm, rotated rx 180 ry 0 rz -180 deg; joints [2.371, 71.015, -37.608, 4.302, -33.481, -3.59]
  Call Extruder 0.00011
  MoveL (T19920) to (116.68, 118.65, 20.1) mm, rotated rx 180 ry 0 rz -180 deg; joints [2.371, 71.015, -37.608, 4.302, -33.481, -3.59]
  Call Extruder 0.00626
  MoveL (T19921) to (122.25, 118.65, 20.1) mm, rotated rx 180 ry 0 rz -180 deg; joints [2.432, 71.022, -37.623, 4.412, -33.478, -3.682]
  Call Extruder 0.00011
  MoveL (T19922) to (122.25, 118.55, 20.1) mm, rotated rx 180 ry 0 rz -180 deg; joints [2.432, 71.022, -37.623, 4.412, -33.478, -3.682]
  Call Extruder 0.00626
  MoveL (T19923) to (116.68, 118.55, 20.1) mm, rotated rx 180 ry 0 rz -180 deg; joints [2.432, 71.022, -37.623, 4.412, -33.478, -3.682]
  Call Extruder 0.00011
  MoveL (T19924) to (116.68, 118.45, 20.1) mm, rotated rx 180 ry 0 rz -180 deg; joints [2.041, 69.796, -35.32, 3.602, -34.529, -2.969]
  Call Extruder 0.00626
  MoveL (T19925) to (122.25, 118.45, 20.1) mm, rotated rx 180 ry 0 rz -180 deg; joints [2.041, 69.796, -35.32, 3.602, -34.529, -2.969]
  Call Extruder 0.00011
  MoveL (T19926) to (122.25, 118.35, 20.1) mm, rotated rx 180 ry 0 rz -180 deg; joints [2.041, 69.796, -35.32, 3.602, -34.529, -2.969]
  Call Extruder 0.00626
  MoveL (T19927) to (116.68, 118.35, 20.1) mm, rotated rx 180 ry 0 rz -180 deg; joints [2.048, 69.778, -35.285, 3.613, -34.546, -2.977]
  Call Extruder 0.00012
  MoveL (T19928) to (116.63, 118.25, 20.1) mm, rotated rx 180 ry 0 rz -180 deg; joints [2.048, 69.778, -35.285, 3.613, -34.546, -2.977]
  Call Extruder 0.00631
  MoveL (T19929) to (122.25, 118.25, 20.1) mm, rotated rx 180 ry 0 rz -180 deg; joints [2.048, 69.778, -35.285, 3.613, -34.546, -2.977]
  Call Extruder 0.00011
  MoveL (T19930) to (122.25, 118.15, 20.1) mm, rotated rx 180 ry 0 rz -180 deg; joints [2.048, 69.778, -35.285, 3.613, -34.546, -2.977]
  Call Extruder 0.00636
  MoveL (T19931) to (116.58, 118.15, 20.1) mm, rotated rx 180 ry 0 rz -180 deg; joints [2.053, 69.772, -35.274, 3.622, -34.551, -2.985]
  Call Extruder 0.00013
  MoveL (T19932) to (116.53, 118.05, 20.1) mm, rotated rx 180 ry 0 rz -180 deg; joints [2.053, 69.772, -35.274, 3.622, -34.551, -2.985]
  Call Extruder 0.00642
  MoveL (T19933) to (122.25, 118.05, 20.1) mm, rotated rx 180 ry 0 rz -180 deg; joints [2.093, 69.776, -35.282, 3.693, -34.55, -3.043]
  Call Extruder 0.00011
  MoveL (T19934) to (122.25, 117.95, 20.1) mm, rotated rx 180 ry 0 rz -180 deg; joints [2.493, 71.03, -37.637, 4.523, -33.475, -3.775]
  Call Extruder 0.00648
  MoveL (T19935) to (116.48, 117.95, 20.1) mm, rotated rx 180 ry 0 rz -180 deg; joints [2.493, 71.03, -37.637, 4.523, -33.475, -3.775]
  Call Extruder 0.00013
  MoveL (T19936) to (116.43, 117.85, 20.1) mm, rotated rx 180 ry 0 rz -180 deg; joints [2.493, 71.03, -37.637, 4.523, -33.475, -3.775]
  Call Extruder 0.00654
  MoveL (T19937) to (122.25, 117.85, 20.1) mm, rotated rx 180 ry 0 rz -180 deg; joints [2.553, 71.038, -37.652, 4.633, -33.472, -3.867]
  Call Extruder 0.00011
  MoveL (T19938) to (122.25, 117.75, 20.1) mm, rotated rx 180 ry 0 rz -180 deg; joints [2.553, 71.038, -37.652, 4.633, -33.472, -3.867]
  Call Extruder 0.00659
  MoveL (T19939) to (116.38, 117.75, 20.1) mm, rotated rx 180 ry 0 rz -180 deg; joints [2.154, 69.782, -35.294, 3.801, -34.548, -3.132]
  Call Extruder 0.00013
  MoveL (T19940) to (116.33, 117.65, 20.1) mm, rotated rx 180 ry 0 rz -180 deg; joints [2.154, 69.782, -35.294, 3.801, -34.548, -3.132]
  Call Extruder 0.00665
  MoveL (T19941) to (122.25, 117.65, 20.1) mm, rotated rx 180 ry 0 rz -180 deg; joints [2.154, 69.782, -35.294, 3.801, -34.548, -3.132]
  Call Extruder 0.00011
  MoveL (T19942) to (122.25, 117.55, 20.1) mm, rotated rx 180 ry 0 rz -180 deg; joints [2.216, 69.789, -35.305, 3.909, -34.546, -3.222]
  Call Extruder 0.00671
  MoveL (T19943) to (116.27, 117.55, 20.1) mm, rotated rx 180 ry 0 rz -180 deg; joints [2.216, 69.789, -35.305, 3.909, -34.546, -3.222]
  Call Extruder 0.00013
  MoveL (T19944) to (116.22, 117.45, 20.1) mm, rotated rx 180 ry 0 rz -180 deg; joints [2.216, 69.789, -35.305, 3.909, -34.546, -3.222]
  Call Extruder 0.00677
  MoveL (T19945) to (122.25, 117.45, 20.1) mm, rotated rx 180 ry 0 rz -180 deg; joints [2.614, 71.046, -37.668, 4.744, -33.469, -3.96]
  Call Extruder 0.00011
  MoveL (T19946) to (122.25, 117.35, 20.1) mm, rotated rx 180 ry 0 rz -180 deg; joints [2.614, 71.046, -37.668, 4.744, -33.469, -3.96]
  Call Extruder 0.00682
  MoveL (T19947) to (116.17, 117.35, 20.1) mm, rotated rx 180 ry 0 rz -180 deg; joints [2.614, 71.046, -37.668, 4.744, -33.469, -3.96]
  Call Extruder 0.00013
  MoveL (T19948) to (116.12, 117.25, 20.1) mm, rotated rx 180 ry 0 rz -180 deg; joints [2.614, 71.046, -37.668, 4.744, -33.469, -3.96]
  Call Extruder 0.00688
  MoveL (T19949) to (122.25, 117.25, 20.1) mm, rotated rx 180 ry 0 rz -180 deg; joints [2.675, 71.055, -37.684, 4.855, -33.466, -4.053]
  Call Extruder 0.00011
  MoveL (T19950) to (122.25, 117.15, 20.1) mm, rotated rx 180 ry 0 rz -180 deg; joints [2.675, 71.055, -37.684, 4.855, -33.466, -4.053]
  Call Extruder 0.00694
  MoveL (T19951) to (116.07, 117.15, 20.1) mm, rotated rx 180 ry 0 rz -180 deg; joints [2.277, 69.795, -35.318, 4.018, -34.543, -3.311]
  Call Extruder 0.00013
  MoveL (T19952) to (116.02, 117.05, 20.1) mm, rotated rx 180 ry 0 rz -180 deg; joints [2.338, 69.802, -35.331, 4.126, -34.541, -3.4]
  Call Extruder 0.007
  MoveL (T19953) to (122.25, 117.05, 20.1) mm, rotated rx 180 ry 0 rz -180 deg; joints [2.338, 69.802, -35.331, 4.126, -34.541, -3.4]
  Call Extruder 0.00011
  MoveL (T19954) to (122.25, 116.95, 20.1) mm, rotated rx 180 ry 0 rz -180 deg; joints [2.71, 70.98, -37.544, 4.91, -33.534, -4.096]
  Call Extruder 0.00705
  MoveL (T19955) to (115.97, 116.95, 20.1) mm, rotated rx 180 ry 0 rz -180 deg; joints [2.71, 70.98, -37.544, 4.91, -33.534, -4.096]
  Call Extruder 0.00013
  MoveL (T19956) to (115.92, 116.85, 20.1) mm, rotated rx 180 ry 0 rz -180 deg; joints [2.71, 70.98, -37.544, 4.91, -33.534, -4.096]
  Call Extruder 0.00711
  MoveL (T19957) to (122.25, 116.85, 20.1) mm, rotated rx 180 ry 0 rz -180 deg; joints [2.71, 70.98, -37.544, 4.91, -33.534, -4.096]
  Call Extruder 0.00011
  MoveL (T19958) to (122.25, 116.75, 20.1) mm, rotated rx 180 ry 0 rz -180 deg; joints [2.713, 70.8, -37.205, 4.895, -33.692, -4.076]
  Call Extruder 0.00717
  MoveL (T19959) to (115.86, 116.75, 20.1) mm, rotated rx 180 ry 0 rz -180 deg; joints [2.713, 70.8, -37.205, 4.895, -33.692, -4.076]
  Call Extruder 0.00013
  MoveL (T19960) to (115.81, 116.65, 20.1) mm, rotated rx 180 ry 0 rz -180 deg; joints [2.399, 69.809, -35.344, 4.234, -34.538, -3.49]
  Call Extruder 0.00723
  MoveL (T19961) to (122.25, 116.65, 20.1) mm, rotated rx 180 ry 0 rz -180 deg; joints [2.46, 69.816, -35.357, 4.342, -34.536, -3.579]
  Call Extruder 0.00011
  MoveL (T19962) to (122.25, 116.55, 20.1) mm, rotated rx 180 ry 0 rz -180 deg; joints [2.46, 69.816, -35.357, 4.342, -34.536, -3.579]
  Call Extruder 0.00728
  MoveL (T19963) to (115.76, 116.55, 20.1) mm, rotated rx 180 ry 0 rz -180 deg; joints [2.46, 69.816, -35.357, 4.342, -34.536, -3.579]
  Call Extruder 0.00013
  MoveL (T19964) to (115.71, 116.45, 20.1) mm, rotated rx 180 ry 0 rz -180 deg; joints [2.716, 70.621, -36.868, 4.88, -33.849, -4.056]
  Call Extruder 0.00734
  MoveL (T19965) to (122.25, 116.45, 20.1) mm, rotated rx 180 ry 0 rz -180 deg; joints [2.716, 70.621, -36.868, 4.88, -33.849, -4.056]
  Call Extruder 0.00011
  MoveL (T19966) to (122.25, 116.35, 20.1) mm, rotated rx 180 ry 0 rz -180 deg; joints [2.719, 70.452, -36.551, 4.866, -33.997, -4.037]
  Call Extruder 0.0074
  MoveL (T19967) to (115.66, 116.35, 20.1) mm, rotated rx 180 ry 0 rz -180 deg; joints [2.719, 70.452, -36.551, 4.866, -33.997, -4.037]
  Call Extruder 0.00013
  MoveL (T19968) to (115.61, 116.25, 20.1) mm, rotated rx 180 ry 0 rz -180 deg; joints [2.719, 70.452, -36.551, 4.866, -33.997, -4.037]
  Call Extruder 0.00745
  MoveL (T19969) to (122.25, 116.25, 20.1) mm, rotated rx 180 ry 0 rz -180 deg; joints [2.717, 70.436, -36.522, 4.861, -34.01, -4.033]
  Call Extruder 0.00011
  MoveL (T19970) to (122.25, 116.15, 20.1) mm, rotated rx 180 ry 0 rz -180 deg; joints [2.717, 70.436, -36.522, 4.861, -34.01, -4.033]
  Call Extruder 0.00751
  MoveL (T19971) to (115.56, 116.15, 20.1) mm, rotated rx 180 ry 0 rz -180 deg; joints [2.503, 69.767, -35.265, 4.412, -34.582, -3.635]
  Call Extruder 0.00013
  MoveL (T19972) to (115.51, 116.05, 20.1) mm, rotated rx 180 ry 0 rz -180 deg; joints [2.503, 69.767, -35.265, 4.412, -34.582, -3.635]
  Call Extruder 0.00757
  MoveL (T19973) to (122.25, 116.05, 20.1) mm, rotated rx 180 ry 0 rz -180 deg; joints [2.503, 69.767, -35.265, 4.412, -34.582, -3.635]
  Call Extruder 0.00011
  MoveL (T19974) to (122.25, 115.95, 20.1) mm, rotated rx 180 ry 0 rz -180 deg; joints [2.503, 69.767, -35.265, 4.412, -34.582, -3.635]
  Call Extruder 0.00763
  MoveL (T19975) to (115.45, 115.95, 20.1) mm, rotated rx 180 ry 0 rz -180 deg; joints [2.503, 69.767, -35.265, 4.412, -34.582, -3.635]
  Call Extruder 0.00013
  MoveL (T19976) to (115.4, 115.85, 20.1) mm, rotated rx 180 ry 0 rz -180 deg; joints [2.579, 70.002, -35.706, 4.57, -34.381, -3.774]
  Call Extruder 0.00768
  MoveL (T19977) to (122.25, 115.85, 20.1) mm, rotated rx 180 ry 0 rz -180 deg; joints [2.579, 70.002, -35.706, 4.57, -34.381, -3.774]
  Call Extruder 0.00011
  MoveL (T19978) to (122.25, 115.75, 20.1) mm, rotated rx 180 ry 0 rz -180 deg; joints [2.579, 70.002, -35.706, 4.57, -34.381, -3.774]
  Call Extruder 0.00774
  MoveL (T19979) to (115.35, 115.75, 20.1) mm, rotated rx 180 ry 0 rz -180 deg; joints [2.579, 70.002, -35.706, 4.57, -34.381, -3.774]
  Call Extruder 0.00013
  MoveL (T19980) to (115.3, 115.65, 20.1) mm, rotated rx 180 ry 0 rz -180 deg; joints [1.869, 68.889, -34.014, 3.266, -34.918, -2.679]
  Call Extruder 0.0078
  MoveL (T19981) to (122.25, 115.65, 20.1) mm, rotated rx 180 ry 0 rz -180 deg; joints [1.869, 69.121, -34.053, 3.25, -35.112, -2.66]
  Call Extruder 0.00011
  MoveL (T19982) to (122.25, 115.55, 20.1) mm, rotated rx 180 ry 0 rz -180 deg; joints [1.869, 69.121, -34.053, 3.25, -35.112, -2.66]
  Call Extruder 0.00786
  MoveL (T19983) to (115.25, 115.55, 20.1) mm, rotated rx 180 ry 0 rz -180 deg; joints [1.869, 69.121, -34.053, 3.25, -35.112, -2.66]
  Call Extruder 0.00013
  MoveL (T19984) to (115.2, 115.45, 20.1) mm, rotated rx 180 ry 0 rz -180 deg; joints [1.869, 69.121, -34.053, 3.25, -35.112, -2.66]
  Call Extruder 0.00791
  MoveL (T19985) to (122.25, 115.45, 20.1) mm, rotated rx 180 ry 0 rz -180 deg; joints [1.869, 69.121, -34.053, 3.25, -35.112, -2.66]
  Call Extruder 0.00011
  MoveL (T19986) to (122.25, 115.35, 20.1) mm, rotated rx 180 ry 0 rz -180 deg; joints [1.869, 69.121, -34.053, 3.25, -35.112, -2.66]
  Call Extruder 0.00797
  MoveL (T19987) to (115.15, 115.35, 20.1) mm, rotated rx 180 ry 0 rz -180 deg; joints [1.869, 69.121, -34.053, 3.25, -35.112, -2.66]
  Call Extruder 0.00013
  MoveL (T19988) to (115.1, 115.25, 20.1) mm, rotated rx 180 ry 0 rz -180 deg; joints [1.869, 69.121, -34.053, 3.25, -35.112, -2.66]
  Call Extruder 0.00803
  MoveL (T19989) to (122.25, 115.25, 20.1) mm, rotated rx 180 ry 0 rz -180 deg; joints [1.874, 68.686, -33.234, 3.229, -35.494, -2.63]
  Call Extruder 0.00011
  MoveL (T19990) to (122.25, 115.15, 20.1) mm, rotated rx 180 ry 0 rz -180 deg; joints [1.874, 68.686, -33.234, 3.229, -35.494, -2.63]
  Call Extruder 0.00809
  MoveL (T19991) to (115.05, 115.15, 20.1) mm, rotated rx 180 ry 0 rz -180 deg; joints [1.866, 68.628, -33.126, 3.211, -35.545, -2.614]
  Call Extruder 0.00013
  MoveL (T19992) to (115, 115.05, 20.1) mm, rotated rx 180 ry 0 rz -180 deg; joints [1.866, 68.628, -33.126, 3.211, -35.545, -2.614]
  Call Extruder 0.00814
  MoveL (T19993) to (122.25, 115.05, 20.1) mm, rotated rx 180 ry 0 rz -180 deg; joints [1.866, 68.628, -33.126, 3.211, -35.545, -2.614]
  Call Extruder 0.00011
  MoveL (T19994) to (122.25, 114.95, 20.1) mm, rotated rx 180 ry 0 rz -180 deg; joints [1.815, 68.483, -32.854, 3.113, -35.669, -2.53]
  Call Extruder 0.0082
  MoveL (T19995) to (114.94, 114.95, 20.1) mm, rotated rx 180 ry 0 rz -180 deg; joints [2.818, 66.166, -28.505, 4.606, -37.751, -3.645]
  Call Extruder 0.00013
  MoveL (T19996) to (114.89, 114.85, 20.1) mm, rotated rx 180 ry 0 rz -180 deg; joints [2.818, 66.166, -28.505, 4.606, -37.751, -3.645]
  Call Extruder 0.00826
  MoveL (T19997) to (122.25, 114.85, 20.1) mm, rotated rx 180 ry 0 rz -180 deg; joints [2.818, 66.166, -28.505, 4.606, -37.751, -3.645]
  Call Extruder 0.00011
  MoveL (T19998) to (122.25, 114.75, 20.1) mm, rotated rx 180 ry 0 rz -180 deg; joints [2.938, 66.18, -28.532, 4.803, -37.746, -3.801]
  Call Extruder 0.00832
  MoveL (T19999) to (114.84, 114.75, 20.1) mm, rotated rx 180 ry 0 rz -180 deg; joints [2.938, 66.18, -28.532, 4.803, -37.746, -3.801]
  Call Extruder 0.00013
  MoveL (T20000) to (114.79, 114.65, 20.1) mm, rotated rx 180 ry 0 rz -180 deg; joints [2.938, 66.18, -28.532, 4.803, -37.746, -3.801]
  Call Extruder 0.00837
  MoveL (T20001) to (122.25, 114.65, 20.1) mm, rotated rx 180 ry 0 rz -180 deg; joints [3.295, 67.146, -30.345, 5.489, -36.928, -4.393]
  Call Extruder 0.00011
  MoveL (T20002) to (122.25, 114.55, 20.1) mm, rotated rx 180 ry 0 rz -180 deg; joints [3.295, 67.146, -30.345, 5.489, -36.928, -4.393]
  Call Extruder 0.00843
  MoveL (T20003) to (114.74, 114.55, 20.1) mm, rotated rx 180 ry 0 rz -180 deg; joints [3.288, 67.445, -30.904, 5.511, -36.667, -4.425]
  Call Extruder 0.00013
  MoveL (T20004) to (114.69, 114.45, 20.1) mm, rotated rx 180 ry 0 rz -180 deg; joints [3.288, 67.445, -30.904, 5.511, -36.667, -4.425]
  Call Extruder 0.00849
  MoveL (T20005) to (122.25, 114.45, 20.1) mm, rotated rx 180 ry 0 rz -180 deg; joints [2.356, 69.683, -35.108, 4.146, -34.646, -3.413]
  Call Extruder 0.00011
  MoveL (T20006) to (122.25, 114.35, 20.1) mm, rotated rx 180 ry 0 rz -180 deg; joints [2.356, 69.683, -35.108, 4.146, -34.646, -3.413]
  Call Extruder 0.00855
  MoveL (T20007) to (114.64, 114.35, 20.1) mm, rotated rx 180 ry 0 rz -180 deg; joints [2.356, 69.683, -35.108, 4.146, -34.646, -3.413]
  Call Extruder 0.00013
  MoveL (T20008) to (114.58, 114.25, 20.1) mm, rotated rx 180 ry 0 rz -180 deg; joints [2.29, 69.676, -35.094, 4.03, -34.648, -3.317]
  Call Extruder 0.0086
  MoveL (T20009) to (122.25, 114.25, 20.1) mm, rotated rx 180 ry 0 rz -180 deg; joints [2.29, 69.676, -35.094, 4.03, -34.648, -3.317]
  Call Extruder 0.00011
  MoveL (T20010) to (122.25, 114.15, 20.1) mm, rotated rx 180 ry 0 rz -180 deg; joints [1.775, 68.184, -32.293, 3.026, -35.929, -2.451]
  Call Extruder 0.00866
  MoveL (T20011) to (114.53, 114.15, 20.1) mm, rotated rx 180 ry 0 rz -180 deg; joints [1.775, 68.184, -32.293, 3.026, -35.929, -2.451]
  Call Extruder 0.00013
  MoveL (T20012) to (114.48, 114.05, 20.1) mm, rotated rx 180 ry 0 rz -180 deg; joints [1.875, 67.942, -31.839, 3.179, -36.146, -2.568]
  Call Extruder 0.00872
  MoveL (T20013) to (122.25, 114.05, 20.1) mm, rotated rx 180 ry 0 rz -180 deg; joints [1.875, 67.942, -31.839, 3.179, -36.146, -2.568]
  Call Extruder 0.00011
  MoveL (T20014) to (122.25, 113.95, 20.1) mm, rotated rx 180 ry 0 rz -180 deg; joints [1.875, 67.942, -31.839, 3.179, -36.146, -2.568]
  Call Extruder 0.00878
  MoveL (T20015) to (114.43, 113.95, 20.1) mm, rotated rx 180 ry 0 rz -180 deg; joints [1.875, 67.942, -31.839, 3.179, -36.146, -2.568]
  Call Extruder 0.00013
  MoveL (T20016) to (114.38, 113.85, 20.1) mm, rotated rx 180 ry 0 rz -180 deg; joints [1.875, 67.942, -31.839, 3.179, -36.146, -2.568]
  Call Extruder 0.00883
  MoveL (T20017) to (122.25, 113.85, 20.1) mm, rotated rx 180 ry 0 rz -180 deg; joints [1.875, 67.942, -31.839, 3.179, -36.146, -2.568]
  Call Extruder 0.00011
  MoveL (T20018) to (122.25, 113.75, 20.1) mm, rotated rx 180 ry 0 rz -180 deg; joints [1.888, 67.629, -31.251, 3.18, -36.421, -2.56]
  Call Extruder 0.00889
  MoveL (T20019) to (114.33, 113.75, 20.1) mm, rotated rx 180 ry 0 rz -180 deg; joints [1.888, 67.629, -31.251, 3.18, -36.421, -2.56]
  Call Extruder 0.00013
  MoveL (T20020) to (114.28, 113.65, 20.1) mm, rotated rx 180 ry 0 rz -180 deg; joints [1.888, 67.629, -31.251, 3.18, -36.421, -2.56]
  Call Extruder 0.00895
  MoveL (T20021) to (122.25, 113.65, 20.1) mm, rotated rx 180 ry 0 rz -180 deg; joints [1.888, 67.629, -31.251, 3.18, -36.421, -2.56]
  Call Extruder 0.00011
  MoveL (T20022) to (122.25, 113.55, 20.1) mm, rotated rx 180 ry 0 rz -180 deg; joints [1.888, 67.629, -31.251, 3.18, -36.421, -2.56]
  Call Extruder 0.00901
  MoveL (T20023) to (114.23, 113.55, 20.1) mm, rotated rx 180 ry 0 rz -180 deg; joints [1.888, 67.629, -31.251, 3.18, -36.421, -2.56]
  Call Extruder 0.00013
  MoveL (T20024) to (114.18, 113.45, 20.1) mm, rotated rx 180 ry 0 rz -180 deg; joints [1.888, 67.629, -31.251, 3.18, -36.421, -2.56]
  Call Extruder 0.00906
  MoveL (T20025) to (122.25, 113.45, 20.1) mm, rotated rx 180 ry 0 rz -180 deg; joints [1.888, 67.629, -31.251, 3.18, -36.421, -2.56]
  Call Extruder 0.00011
  MoveL (T20026) to (122.25, 113.35, 20.1) mm, rotated rx 180 ry 0 rz -180 deg; joints [1.888, 67.629, -31.251, 3.18, -36.421, -2.56]
  Call Extruder 0.00912
  MoveL (T20027) to (114.12, 113.35, 20.1) mm, rotated rx 180 ry 0 rz -180 deg; joints [1.888, 67.629, -31.251, 3.18, -36.421, -2.56]
  Call Extruder 0.00013
  MoveL (T20028) to (114.07, 113.25, 20.1) mm, rotated rx 180 ry 0 rz -180 deg; joints [1.884, 67.888, -31.736, 3.192, -36.194, -2.577]
  Call Extruder 0.00918
  MoveL (T20029) to (122.25, 113.25, 20.1) mm, rotated rx 180 ry 0 rz -180 deg; joints [1.884, 67.888, -31.736, 3.192, -36.194, -2.577]
  Call Extruder 0.00011
  MoveL (T20030) to (122.25, 113.15, 20.1) mm, rotated rx 180 ry 0 rz -180 deg; joints [1.879, 67.918, -31.793, 3.185, -36.167, -2.572]
  Call Extruder 0.00924
  MoveL (T20031) to (114.02, 113.15, 20.1) mm, rotated rx 180 ry 0 rz -180 deg; joints [1.879, 67.918, -31.793, 3.185, -36.167, -2.572]
  Call Extruder 0.00013
  MoveL (T20032) to (113.97, 113.05, 20.1) mm, rotated rx 180 ry 0 rz -180 deg; joints [1.879, 67.918, -31.793, 3.185, -36.167, -2.572]
  Call Extruder 0.00929
  MoveL (T20033) to (122.25, 113.05, 20.1) mm, rotated rx 180 ry 0 rz -180 deg; joints [1.879, 67.918, -31.793, 3.185, -36.167, -2.572]
  Call Extruder 0.00011
  MoveL (T20034) to (122.25, 112.95, 20.1) mm, rotated rx 180 ry 0 rz -180 deg; joints [1.879, 67.918, -31.793, 3.185, -36.167, -2.572]
  Call Extruder 0.00935
  MoveL (T20035) to (113.92, 112.95, 20.1) mm, rotated rx 180 ry 0 rz -180 deg; joints [1.879, 67.918, -31.793, 3.185, -36.167, -2.572]
  Call Extruder 0.00013
  MoveL (T20036) to (113.87, 112.85, 20.1) mm, rotated rx 180 ry 0 rz -180 deg; joints [1.879, 67.684, -31.756, 3.2, -35.971, -2.591]
  Call Extruder 0.00941
  MoveL (T20037) to (122.25, 112.85, 20.1) mm, rotated rx 180 ry 0 rz -180 deg; joints [1.476, 70.42, -36.886, 2.67, -33.563, -2.225]
  Call Extruder 0.00011
  MoveL (T20038) to (122.25, 112.75, 20.1) mm, rotated rx 180 ry 0 rz -180 deg; joints [1.476, 70.652, -36.926, 2.657, -33.754, -2.209]
  Call Extruder 0.00947
  MoveL (T20039) to (113.82, 112.75, 20.1) mm, rotated rx 180 ry 0 rz -180 deg; joints [1.476, 70.652, -36.926, 2.657, -33.754, -2.209]
  Call Extruder 0.00013
  MoveL (T20040) to (113.77, 112.65, 20.1) mm, rotated rx 180 ry 0 rz -180 deg; joints [1.476, 70.652, -36.926, 2.657, -33.754, -2.209]
  Call Extruder 0.00952
  MoveL (T20041) to (122.25, 112.65, 20.1) mm, rotated rx 180 ry 0 rz -180 deg; joints [1.476, 70.652, -36.926, 2.657, -33.754, -2.209]
  Call Extruder 0.00011
  MoveL (T20042) to (122.25, 112.55, 20.1) mm, rotated rx 180 ry 0 rz -180 deg; joints [1.476, 70.652, -36.926, 2.657, -33.754, -2.209]
  Call Extruder 0.00958
  MoveL (T20043) to (113.72, 112.55, 20.1) mm, rotated rx 180 ry 0 rz -180 deg; joints [1.476, 70.652, -36.926, 2.657, -33.754, -2.209]
  Call Extruder 0.00013
  MoveL (T20044) to (113.66, 112.45, 20.1) mm, rotated rx 180 ry 0 rz -180 deg; joints [1.476, 70.652, -36.926, 2.657, -33.754, -2.209]
  Call Extruder 0.00964
  MoveL (T20045) to (122.25, 112.45, 20.1) mm, rotated rx 180 ry 0 rz -180 deg; joints [1.476, 70.652, -36.926, 2.657, -33.754, -2.209]
  Call Extruder 0.00011
  MoveL (T20046) to (122.25, 112.35, 20.1) mm, rotated rx 180 ry 0 rz -180 deg; joints [1.476, 70.652, -36.926, 2.657, -33.754, -2.209]
  Call Extruder 0.0097
  MoveL (T20047) to (113.61, 112.35, 20.1) mm, rotated rx 180 ry 0 rz -180 deg; joints [1.476, 70.652, -36.926, 2.657, -33.754, -2.209]
  Call Extruder 0.00013
  MoveL (T20048) to (113.56, 112.25, 20.1) mm, rotated rx 180 ry 0 rz -180 deg; joints [1.4, 70.419, -36.49, 2.507, -33.955, -2.08]
  Call Extruder 0.00975
  MoveL (T20049) to (122.25, 112.25, 20.1) mm, rotated rx 180 ry 0 rz -180 deg; joints [1.4, 70.419, -36.49, 2.507, -33.955, -2.08]
  Call Extruder 0.00011
  MoveL (T20050) to (122.25, 112.15, 20.1) mm, rotated rx 180 ry 0 rz -180 deg; joints [1.402, 70.239, -36.151, 2.5, -34.113, -2.07]
  Call Extruder 0.00981
  MoveL (T20051) to (113.51, 112.15, 20.1) mm, rotated rx 180 ry 0 rz -180 deg; joints [1.402, 70.239, -36.151, 2.5, -34.113, -2.07]
  Call Extruder 0.00013
  MoveL (T20052) to (113.46, 112.05, 20.1) mm, rotated rx 180 ry 0 rz -180 deg; joints [1.402, 70.239, -36.151, 2.5, -34.113, -2.07]
  Call Extruder 0.00987
  MoveL (T20053) to (122.25, 112.05, 20.1) mm, rotated rx 180 ry 0 rz -180 deg; joints [1.402, 70.239, -36.151, 2.5, -34.113, -2.07]
  Call Extruder 0.00011
  MoveL (T20054) to (122.25, 111.95, 20.1) mm, rotated rx 180 ry 0 rz -180 deg; joints [1.52, 70.598, -36.826, 2.732, -33.802, -2.271]
  Call Extruder 0.00992
  MoveL (T20055) to (113.41, 111.95, 20.1) mm, rotated rx 180 ry 0 rz -180 deg; joints [1.52, 70.598, -36.826, 2.732, -33.802, -2.271]
  Call Extruder 0.00013
  MoveL (T20056) to (113.36, 111.85, 20.1) mm, rotated rx 180 ry 0 rz -180 deg; joints [1.582, 70.603, -36.835, 2.844, -33.8, -2.364]
  Call Extruder 0.00998
  MoveL (T20057) to (122.25, 111.85, 20.1) mm, rotated rx 180 ry 0 rz -180 deg; joints [1.582, 70.603, -36.835, 2.844, -33.8, -2.364]
  Call Extruder 0.00011
  MoveL (T20058) to (122.25, 111.75, 20.1) mm, rotated rx 180 ry 0 rz -180 deg; joints [1.582, 70.603, -36.835, 2.844, -33.8, -2.364]
  Call Extruder 0.01004
  MoveL (T20059) to (113.31, 111.75, 20.1) mm, rotated rx 180 ry 0 rz -180 deg; joints [1.403, 70.06, -35.814, 2.492, -34.27, -2.06]
  Call Extruder 0.00013
  MoveL (T20060) to (113.25, 111.65, 20.1) mm, rotated rx 180 ry 0 rz -180 deg; joints [1.403, 70.06, -35.814, 2.492, -34.27, -2.06]
  Call Extruder 0.0101
  MoveL (T20061) to (122.25, 111.65, 20.1) mm, rotated rx 180 ry 0 rz -180 deg; joints [1.403, 70.06, -35.814, 2.492, -34.27, -2.06]
  Call Extruder 0.00011
  MoveL (T20062) to (122.25, 111.55, 20.1) mm, rotated rx 180 ry 0 rz -180 deg; joints [1.405, 69.882, -35.48, 2.485, -34.427, -2.05]
  Call Extruder 0.01015
  MoveL (T20063) to (113.2, 111.55, 20.1) mm, rotated rx 180 ry 0 rz -180 deg; joints [1.405, 69.882, -35.48, 2.485, -34.427, -2.05]
  Call Extruder 0.00013
  MoveL (T20064) to (113.15, 111.45, 20.1) mm, rotated rx 180 ry 0 rz -180 deg; joints [1.405, 69.882, -35.48, 2.485, -34.427, -2.05]
  Call Extruder 0.01021
  MoveL (T20065) to (122.25, 111.45, 20.1) mm, rotated rx 180 ry 0 rz -180 deg; joints [1.405, 69.882, -35.48, 2.485, -34.427, -2.05]
  Call Extruder 0.00011
  MoveL (T20066) to (122.25, 111.35, 20.1) mm, rotated rx 180 ry 0 rz -180 deg; joints [1.405, 69.882, -35.48, 2.485, -34.427, -2.05]
  Call Extruder 0.01027
  MoveL (T20067) to (113.1, 111.35, 20.1) mm, rotated rx 180 ry 0 rz -180 deg; joints [1.624, 70.545, -36.727, 2.916, -33.853, -2.422]
  Call Extruder 0.00013
  MoveL (T20068) to (113.05, 111.25, 20.1) mm, rotated rx 180 ry 0 rz -180 deg; joints [1.656, 70.457, -36.561, 2.968, -33.932, -2.463]
  Call Extruder 0.01033
  MoveL (T20069) to (122.25, 111.25, 20.1) mm, rotated rx 180 ry 0 rz -180 deg; joints [1.656, 70.457, -36.561, 2.968, -33.932, -2.463]
  Call Extruder 0.00011
  MoveL (T20070) to (122.25, 111.15, 20.1) mm, rotated rx 180 ry 0 rz -180 deg; joints [1.406, 69.705, -35.149, 2.478, -34.581, -2.041]
  Call Extruder 0.01038
  MoveL (T20071) to (113, 111.15, 20.1) mm, rotated rx 180 ry 0 rz -180 deg; joints [1.406, 69.705, -35.149, 2.478, -34.581, -2.041]
  Call Extruder 0.00013
  MoveL (T20072) to (112.95, 111.05, 20.1) mm, rotated rx 180 ry 0 rz -180 deg; joints [1.406, 69.705, -35.149, 2.478, -34.581, -2.041]
  Call Extruder 0.01044
  MoveL (T20073) to (122.25, 111.05, 20.1) mm, rotated rx 180 ry 0 rz -180 deg; joints [1.408, 69.53, -34.82, 2.471, -34.735, -2.031]
  Call Extruder 0.00011
  MoveL (T20074) to (122.25, 110.95, 20.1) mm, rotated rx 180 ry 0 rz -180 deg; joints [1.408, 69.53, -34.82, 2.471, -34.735, -2.031]
  Call Extruder 0.0105
  MoveL (T20075) to (112.9, 110.95, 20.1) mm, rotated rx 180 ry 0 rz -180 deg; joints [1.408, 69.53, -34.82, 2.471, -34.735, -2.031]
  Call Extruder 0.00013
  MoveL (T20076) to (112.85, 110.85, 20.1) mm, rotated rx 180 ry 0 rz -180 deg; joints [1.408, 69.53, -34.82, 2.471, -34.735, -2.031]
  Call Extruder 0.01056
  MoveL (T20077) to (122.25, 110.85, 20.1) mm, rotated rx 180 ry 0 rz -180 deg; joints [1.688, 70.369, -36.395, 3.019, -34.011, -2.503]
  Call Extruder 0.00011
  MoveL (T20078) to (122.25, 110.75, 20.1) mm, rotated rx 180 ry 0 rz -180 deg; joints [1.688, 70.369, -36.395, 3.019, -34.011, -2.503]
  Call Extruder 0.01061
  MoveL (T20079) to (112.79, 110.75, 20.1) mm, rotated rx 180 ry 0 rz -180 deg; joints [1.688, 70.369, -36.395, 3.019, -34.011, -2.503]
  Call Extruder 0.00013
  MoveL (T20080) to (112.74, 110.65, 20.1) mm, rotated rx 180 ry 0 rz -180 deg; joints [1.72, 70.281, -36.231, 3.07, -34.089, -2.544]
  Call Extruder 0.01067
  MoveL (T20081) to (122.25, 110.65, 20.1) mm, rotated rx 180 ry 0 rz -180 deg; joints [1.72, 70.281, -36.231, 3.07, -34.089, -2.544]
  Call Extruder 0.00011
  MoveL (T20082) to (122.25, 110.55, 20.1) mm, rotated rx 180 ry 0 rz -180 deg; joints [1.72, 70.281, -36.231, 3.07, -34.089, -2.544]
  Call Extruder 0.01073
  MoveL (T20083) to (112.69, 110.55, 20.1) mm, rotated rx 180 ry 0 rz -180 deg; joints [1.72, 70.281, -36.231, 3.07, -34.089, -2.544]
  Call Extruder 0.00013
  MoveL (T20084) to (112.64, 110.45, 20.1) mm, rotated rx 180 ry 0 rz -180 deg; joints [1.409, 69.357, -34.494, 2.465, -34.887, -2.022]
  Call Extruder 0.01079
  MoveL (T20085) to (122.25, 110.45, 20.1) mm, rotated rx 180 ry 0 rz -180 deg; joints [1.409, 69.357, -34.494, 2.465, -34.887, -2.022]
  Call Extruder 0.00011
  MoveL (T20086) to (122.25, 110.35, 20.1) mm, rotated rx 180 ry 0 rz -180 deg; joints [1.409, 69.357, -34.494, 2.465, -34.887, -2.022]
  Call Extruder 0.01084
  MoveL (T20087) to (112.59, 110.35, 20.1) mm, rotated rx 180 ry 0 rz -180 deg; joints [1.409, 69.357, -34.494, 2.465, -34.887, -2.022]
  Call Extruder 0.00013
  MoveL (T20088) to (112.54, 110.25, 20.1) mm, rotated rx 180 ry 0 rz -180 deg; joints [1.411, 69.184, -34.17, 2.458, -35.039, -2.013]
  Call Extruder 0.0109
  MoveL (T20089) to (122.25, 110.25, 20.1) mm, rotated rx 180 ry 0 rz -180 deg; joints [1.411, 69.184, -34.17, 2.458, -35.039, -2.013]
  Call Extruder 0.00011
  MoveL (T20090) to (122.25, 110.15, 20.1) mm, rotated rx 180 ry 0 rz -180 deg; joints [1.411, 69.184, -34.17, 2.458, -35.039, -2.013]
  Call Extruder 0.01096
  MoveL (T20091) to (112.49, 110.15, 20.1) mm, rotated rx 180 ry 0 rz -180 deg; joints [1.753, 70.194, -36.067, 3.122, -34.166, -2.584]
  Call Extruder 0.00013
  MoveL (T20092) to (112.44, 110.05, 20.1) mm, rotated rx 180 ry 0 rz -180 deg; joints [1.753, 70.194, -36.067, 3.122, -34.166, -2.584]
  Call Extruder 0.01102
  MoveL (T20093) to (122.25, 110.05, 20.1) mm, rotated rx 180 ry 0 rz -180 deg; joints [1.753, 70.194, -36.067, 3.122, -34.166, -2.584]
  Call Extruder 0.00011
  MoveL (T20094) to (122.25, 109.95, 20.1) mm, rotated rx 180 ry 0 rz -180 deg; joints [1.785, 70.107, -35.904, 3.173, -34.244, -2.624]
  Call Extruder 0.01107
  MoveL (T20095) to (112.39, 109.95, 20.1) mm, rotated rx 180 ry 0 rz -180 deg; joints [1.785, 70.107, -35.904, 3.173, -34.244, -2.624]
  Call Extruder 0.00013
  MoveL (T20096) to (112.33, 109.85, 20.1) mm, rotated rx 180 ry 0 rz -180 deg; joints [1.412, 69.013, -33.848, 2.451, -35.189, -2.004]
  Call Extruder 0.01113
  MoveL (T20097) to (122.25, 109.85, 20.1) mm, rotated rx 180 ry 0 rz -180 deg; joints [1.412, 69.013, -33.848, 2.451, -35.189, -2.004]
  Call Extruder 0.00011
  MoveL (T20098) to (122.25, 109.75, 20.1) mm, rotated rx 180 ry 0 rz -180 deg; joints [1.414, 68.843, -33.529, 2.445, -35.338, -1.995]
  Call Extruder 0.01119
  MoveL (T20099) to (112.28, 109.75, 20.1) mm, rotated rx 180 ry 0 rz -180 deg; joints [1.414, 68.843, -33.529, 2.445, -35.338, -1.995]
  Call Extruder 0.00013
  MoveL (T20100) to (112.23, 109.65, 20.1) mm, rotated rx 180 ry 0 rz -180 deg; joints [1.414, 68.843, -33.529, 2.445, -35.338, -1.995]
  Call Extruder 0.01125
  MoveL (T20101) to (122.25, 109.65, 20.1) mm, rotated rx 180 ry 0 rz -180 deg; joints [1.815, 70.016, -35.732, 3.221, -34.326, -2.661]
  Call Extruder 0.00011
  MoveL (T20102) to (122.25, 109.55, 20.1) mm, rotated rx 180 ry 0 rz -180 deg; joints [1.815, 70.016, -35.732, 3.221, -34.326, -2.661]
  Call Extruder 0.0113
  MoveL (T20103) to (112.18, 109.55, 20.1) mm, rotated rx 180 ry 0 rz -180 deg; joints [1.815, 70.016, -35.732, 3.221, -34.326, -2.661]
  Call Extruder 0.00013
